SetDO drillDone,1;
WaitUntil drillDone = 0;
        MoveL RelTool(Target_3860,0,0,-10),v30,z10,DrillTool\WObj:=FakeWing;
        MoveL RelTool(Target_3870,0,0,-10),v30,z10,DrillTool\WObj:=FakeWing;
        MoveL Target_3870,v30,fine,DrillTool\WObj:=FakeWing;
SetDO drillDone,1;
WaitUntil drillDone = 0;
        MoveL RelTool(Target_3870,0,0,-10),v30,z10,DrillTool\WObj:=FakeWing;
        MoveL RelTool(Target_3880,0,0,-10),v30,z10,DrillTool\WObj:=FakeWing;
        MoveL Target_3880,v30,fine,DrillTool\WObj:=FakeWing;
SetDO drillDone,1;
WaitUntil drillDone = 0;
        MoveL RelTool(Target_3880,0,0,-10),v30,z10,DrillTool\WObj:=FakeWing;
        MoveL RelTool(Target_3890,0,0,-10),v30,z10,DrillTool\WObj:=FakeWing;
        MoveL Target_3890,v30,fine,DrillTool\WObj:=FakeWing;
SetDO drillDone,1;
WaitUntil drillDone = 0;
        MoveL RelTool(Target_3890,0,0,-10),v30,z10,DrillTool\WObj:=FakeWing;
        MoveL RelTool(Target_3900,0,0,-10),v30,z10,DrillTool\WObj:=FakeWing;
        MoveL Target_3900,v30,fine,DrillTool\WObj:=FakeWing;
SetDO drillDone,1;
WaitUntil drillDone = 0;
        MoveL RelTool(Target_3900,0,0,-10),v30,z10,DrillTool\WObj:=FakeWing;
        MoveL RelTool(Target_3910,0,0,-10),v30,z10,DrillTool\WObj:=FakeWing;
        MoveL Target_3910,v30,fine,DrillTool\WObj:=FakeWing;
SetDO drillDone,1;
WaitUntil drillDone = 0;
        MoveL RelTool(Target_3910,0,0,-10),v30,z10,DrillTool\WObj:=FakeWing;
        MoveL RelTool(Target_3920,0,0,-10),v30,z10,DrillTool\WObj:=FakeWing;
        MoveL Target_3920,v30,fine,DrillTool\WObj:=FakeWing;
SetDO drillDone,1;
WaitUntil drillDone = 0;
        MoveL RelTool(Target_3920,0,0,-10),v30,z10,DrillTool\WObj:=FakeWing;
        MoveL RelTool(Target_3930,0,0,-10),v30,z10,DrillTool\WObj:=FakeWing;
        MoveL Target_3930,v30,fine,DrillTool\WObj:=FakeWing;
SetDO drillDone,1;
WaitUntil drillDone = 0;
        MoveL RelTool(Target_3930,0,0,-10),v30,z10,DrillTool\WObj:=FakeWing;
        MoveL RelTool(Target_3940,0,0,-10),v30,z10,DrillTool\WObj:=FakeWing;
        MoveL Target_3940,v30,fine,DrillTool\WObj:=FakeWing;
SetDO drillDone,1;
WaitUntil drillDone = 0;
        MoveL RelTool(Target_3940,0,0,-10),v30,z10,DrillTool\WObj:=FakeWing;
        MoveL RelTool(Target_3950,0,0,-10),v30,z10,DrillTool\WObj:=FakeWing;
        MoveL Target_3950,v30,fine,DrillTool\WObj:=FakeWing;
SetDO drillDone,1;
WaitUntil drillDone = 0;
        MoveL RelTool(Target_3950,0,0,-10),v30,z10,DrillTool\WObj:=FakeWing;
        MoveL RelTool(Target_3960,0,0,-10),v30,z10,DrillTool\WObj:=FakeWing;
        MoveL Target_3960,v30,fine,DrillTool\WObj:=FakeWing;
SetDO drillDone,1;
WaitUntil drillDone = 0;
        MoveL RelTool(Target_3960,0,0,-10),v30,z10,DrillTool\WObj:=FakeWing;
        MoveL RelTool(Target_3970,0,0,-10),v30,z10,DrillTool\WObj:=FakeWing;
        MoveL Target_3970,v30,fine,DrillTool\WObj:=FakeWing;
SetDO drillDone,1;
WaitUntil drillDone = 0;
        MoveL RelTool(Target_3970,0,0,-10),v30,z10,DrillTool\WObj:=FakeWing;
        MoveL RelTool(Target_3980,0,0,-10),v30,z10,DrillTool\WObj:=FakeWing;
        MoveL Target_3980,v30,fine,DrillTool\WObj:=FakeWing;
SetDO drillDone,1;
WaitUntil drillDone = 0;
        MoveL RelTool(Target_3980,0,0,-10),v30,z10,DrillTool\WObj:=FakeWing;
        MoveL RelTool(Target_3990,0,0,-10),v30,z10,DrillTool\WObj:=FakeWing;
        MoveL Target_3990,v30,fine,DrillTool\WObj:=FakeWing;
SetDO drillDone,1;
WaitUntil drillDone = 0;
        MoveL RelTool(Target_3990,0,0,-10),v30,z10,DrillTool\WObj:=FakeWing;
        MoveL RelTool(Target_4000,0,0,-10),v30,z10,DrillTool\WObj:=FakeWing;
        MoveL Target_4000,v30,fine,DrillTool\WObj:=FakeWing;
SetDO drillDone,1;
WaitUntil drillDone = 0;
        MoveL RelTool(Target_4000,0,0,-10),v30,z10,DrillTool\WObj:=FakeWing;
        MoveL RelTool(Target_4010,0,0,-10),v30,z10,DrillTool\WObj:=FakeWing;
        MoveL Target_4010,v30,fine,DrillTool\WObj:=FakeWing;
SetDO drillDone,1;
WaitUntil drillDone = 0;
        MoveL RelTool(Target_4010,0,0,-10),v30,z10,DrillTool\WObj:=FakeWing;
        MoveL RelTool(Target_4020,0,0,-10),v30,z10,DrillTool\WObj:=FakeWing;
        MoveL Target_4020,v30,fine,DrillTool\WObj:=FakeWing;
SetDO drillDone,1;
WaitUntil drillDone = 0;
        MoveL RelTool(Target_4020,0,0,-10),v30,z10,DrillTool\WObj:=FakeWing;
        MoveL RelTool(Target_4030,0,0,-10),v30,z10,DrillTool\WObj:=FakeWing;
        MoveL Target_4030,v30,fine,DrillTool\WObj:=FakeWing;
SetDO drillDone,1;
WaitUntil drillDone = 0;
        MoveL RelTool(Target_4030,0,0,-10),v30,z10,DrillTool\WObj:=FakeWing;
        MoveL RelTool(Target_4040,0,0,-10),v30,z10,DrillTool\WObj:=FakeWing;
        MoveL Target_4040,v30,fine,DrillTool\WObj:=FakeWing;
SetDO drillDone,1;
WaitUntil drillDone = 0;
        MoveL RelTool(Target_4040,0,0,-10),v30,z10,DrillTool\WObj:=FakeWing;
        MoveL RelTool(Target_4050,0,0,-10),v30,z10,DrillTool\WObj:=FakeWing;
        MoveL Target_4050,v30,fine,DrillTool\WObj:=FakeWing;
SetDO drillDone,1;
WaitUntil drillDone = 0;
        MoveL RelTool(Target_4050,0,0,-10),v30,z10,DrillTool\WObj:=FakeWing;
        MoveL RelTool(Target_4060,0,0,-10),v30,z10,DrillTool\WObj:=FakeWing;
        MoveL Target_4060,v30,fine,DrillTool\WObj:=FakeWing;
SetDO drillDone,1;
WaitUntil drillDone = 0;
        MoveL RelTool(Target_4060,0,0,-10),v30,z10,DrillTool\WObj:=FakeWing;
        MoveL RelTool(Target_4070,0,0,-10),v30,z10,DrillTool\WObj:=FakeWing;
        MoveL Target_4070,v30,fine,DrillTool\WObj:=FakeWing;
SetDO drillDone,1;
WaitUntil drillDone = 0;
        MoveL RelTool(Target_4070,0,0,-10),v30,z10,DrillTool\WObj:=FakeWing;
        MoveL RelTool(Target_4080,0,0,-10),v30,z10,DrillTool\WObj:=FakeWing;
        MoveL Target_4080,v30,fine,DrillTool\WObj:=FakeWing;
SetDO drillDone,1;
WaitUntil drillDone = 0;
        MoveL RelTool(Target_4080,0,0,-10),v30,z10,DrillTool\WObj:=FakeWing;
        MoveL RelTool(Target_4090,0,0,-10),v30,z10,DrillTool\WObj:=FakeWing;
        MoveL Target_4090,v30,fine,DrillTool\WObj:=FakeWing;
SetDO drillDone,1;
WaitUntil drillDone = 0;
        MoveL RelTool(Target_4090,0,0,-10),v30,z10,DrillTool\WObj:=FakeWing;
        MoveL RelTool(Target_4100,0,0,-10),v30,z10,DrillTool\WObj:=FakeWing;
        MoveL Target_4100,v30,fine,DrillTool\WObj:=FakeWing;
SetDO drillDone,1;
WaitUntil drillDone = 0;
        MoveL RelTool(Target_4100,0,0,-10),v30,z10,DrillTool\WObj:=FakeWing;
        MoveL RelTool(Target_4110,0,0,-10),v30,z10,DrillTool\WObj:=FakeWing;
        MoveL Target_4110,v30,fine,DrillTool\WObj:=FakeWing;
SetDO drillDone,1;
WaitUntil drillDone = 0;
        MoveL RelTool(Target_4110,0,0,-10),v30,z10,DrillTool\WObj:=FakeWing;
        MoveL RelTool(Target_4120,0,0,-10),v30,z10,DrillTool\WObj:=FakeWing;
        MoveL Target_4120,v30,fine,DrillTool\WObj:=FakeWing;
SetDO drillDone,1;
WaitUntil drillDone = 0;
        MoveL RelTool(Target_4120,0,0,-10),v30,z10,DrillTool\WObj:=FakeWing;
        MoveL RelTool(Target_4130,0,0,-10),v30,z10,DrillTool\WObj:=FakeWing;
        MoveL Target_4130,v30,fine,DrillTool\WObj:=FakeWing;
SetDO drillDone,1;
WaitUntil drillDone = 0;
        MoveL RelTool(Target_4130,0,0,-10),v30,z10,DrillTool\WObj:=FakeWing;
        MoveL RelTool(Target_4140,0,0,-10),v30,z10,DrillTool\WObj:=FakeWing;
        MoveL Target_4140,v30,fine,DrillTool\WObj:=FakeWing;
SetDO drillDone,1;
WaitUntil drillDone = 0;
        MoveL RelTool(Target_4140,0,0,-10),v30,z10,DrillTool\WObj:=FakeWing;
        MoveL RelTool(Target_4150,0,0,-10),v30,z10,DrillTool\WObj:=FakeWing;
        MoveL Target_4150,v30,fine,DrillTool\WObj:=FakeWing;
SetDO drillDone,1;
WaitUntil drillDone = 0;
        MoveL RelTool(Target_4150,0,0,-10),v30,z10,DrillTool\WObj:=FakeWing;
        MoveL RelTool(Target_4160,0,0,-10),v30,z10,DrillTool\WObj:=FakeWing;
        MoveL Target_4160,v30,fine,DrillTool\WObj:=FakeWing;
SetDO drillDone,1;
WaitUntil drillDone = 0;
        MoveL RelTool(Target_4160,0,0,-10),v30,z10,DrillTool\WObj:=FakeWing;
        MoveL RelTool(Target_4170,0,0,-10),v30,z10,DrillTool\WObj:=FakeWing;
        MoveL Target_4170,v30,fine,DrillTool\WObj:=FakeWing;
SetDO drillDone,1;
WaitUntil drillDone = 0;
        MoveL RelTool(Target_4170,0,0,-10),v30,z10,DrillTool\WObj:=FakeWing;
        MoveL RelTool(Target_4180,0,0,-10),v30,z10,DrillTool\WObj:=FakeWing;
        MoveL Target_4180,v30,fine,DrillTool\WObj:=FakeWing;
SetDO drillDone,1;
WaitUntil drillDone = 0;
        MoveL RelTool(Target_4180,0,0,-10),v30,z10,DrillTool\WObj:=FakeWing;
        MoveL RelTool(Target_4190,0,0,-10),v30,z10,DrillTool\WObj:=FakeWing;
        MoveL Target_4190,v30,fine,DrillTool\WObj:=FakeWing;
SetDO drillDone,1;
WaitUntil drillDone = 0;
        MoveL RelTool(Target_4190,0,0,-10),v30,z10,DrillTool\WObj:=FakeWing;
        MoveL RelTool(Target_4200,0,0,-10),v30,z10,DrillTool\WObj:=FakeWing;
        MoveL Target_4200,v30,fine,DrillTool\WObj:=FakeWing;
SetDO drillDone,1;
WaitUntil drillDone = 0;
        MoveL RelTool(Target_4200,0,0,-10),v30,z10,DrillTool\WObj:=FakeWing;
        MoveL RelTool(Target_4210,0,0,-10),v30,z10,DrillTool\WObj:=FakeWing;
        MoveL Target_4210,v30,fine,DrillTool\WObj:=FakeWing;
SetDO drillDone,1;
WaitUntil drillDone = 0;
        MoveL RelTool(Target_4210,0,0,-10),v30,z10,DrillTool\WObj:=FakeWing;
        MoveL RelTool(Target_4220,0,0,-10),v30,z10,DrillTool\WObj:=FakeWing;
        MoveL Target_4220,v30,fine,DrillTool\WObj:=FakeWing;
SetDO drillDone,1;
WaitUntil drillDone = 0;
        MoveL RelTool(Target_4220,0,0,-10),v30,z10,DrillTool\WObj:=FakeWing;
        MoveL RelTool(Target_4230,0,0,-10),v30,z10,DrillTool\WObj:=FakeWing;
        MoveL Target_4230,v30,fine,DrillTool\WObj:=FakeWing;
SetDO drillDone,1;
WaitUntil drillDone = 0;
        MoveL RelTool(Target_4230,0,0,-10),v30,z10,DrillTool\WObj:=FakeWing;
        MoveL RelTool(Target_4240,0,0,-10),v30,z10,DrillTool\WObj:=FakeWing;
        MoveL Target_4240,v30,fine,DrillTool\WObj:=FakeWing;
SetDO drillDone,1;
WaitUntil drillDone = 0;
        MoveL RelTool(Target_4240,0,0,-10),v30,z10,DrillTool\WObj:=FakeWing;
        MoveL RelTool(Target_4250,0,0,-10),v30,z10,DrillTool\WObj:=FakeWing;
        MoveL Target_4250,v30,fine,DrillTool\WObj:=FakeWing;
SetDO drillDone,1;
WaitUntil drillDone = 0;
        MoveL RelTool(Target_4250,0,0,-10),v30,z10,DrillTool\WObj:=FakeWing;
        MoveL RelTool(Target_4260,0,0,-10),v30,z10,DrillTool\WObj:=FakeWing;
        MoveL Target_4260,v30,fine,DrillTool\WObj:=FakeWing;
SetDO drillDone,1;
WaitUntil drillDone = 0;
        MoveL RelTool(Target_4260,0,0,-10),v30,z10,DrillTool\WObj:=FakeWing;
        MoveL RelTool(Target_4270,0,0,-10),v30,z10,DrillTool\WObj:=FakeWing;
        MoveL Target_4270,v30,fine,DrillTool\WObj:=FakeWing;
SetDO drillDone,1;
WaitUntil drillDone = 0;
        MoveL RelTool(Target_4270,0,0,-10),v30,z10,DrillTool\WObj:=FakeWing;
        MoveL RelTool(Target_4280,0,0,-10),v30,z10,DrillTool\WObj:=FakeWing;
        MoveL Target_4280,v30,fine,DrillTool\WObj:=FakeWing;
SetDO drillDone,1;
WaitUntil drillDone = 0;
        MoveL RelTool(Target_4280,0,0,-10),v30,z10,DrillTool\WObj:=FakeWing;
        MoveL RelTool(Target_4290,0,0,-10),v30,z10,DrillTool\WObj:=FakeWing;
        MoveL Target_4290,v30,fine,DrillTool\WObj:=FakeWing;
SetDO drillDone,1;
WaitUntil drillDone = 0;
        MoveL RelTool(Target_4290,0,0,-10),v30,z10,DrillTool\WObj:=FakeWing;
        MoveL RelTool(Target_4300,0,0,-10),v30,z10,DrillTool\WObj:=FakeWing;
        MoveL Target_4300,v30,fine,DrillTool\WObj:=FakeWing;
SetDO drillDone,1;
WaitUntil drillDone = 0;
        MoveL RelTool(Target_4300,0,0,-10),v30,z10,DrillTool\WObj:=FakeWing;
        MoveL RelTool(Target_4310,0,0,-10),v30,z10,DrillTool\WObj:=FakeWing;
        MoveL Target_4310,v30,fine,DrillTool\WObj:=FakeWing;
SetDO drillDone,1;
WaitUntil drillDone = 0;
        MoveL RelTool(Target_4310,0,0,-10),v30,z10,DrillTool\WObj:=FakeWing;
        MoveL RelTool(Target_4320,0,0,-10),v30,z10,DrillTool\WObj:=FakeWing;
        MoveL Target_4320,v30,fine,DrillTool\WObj:=FakeWing;
SetDO drillDone,1;
WaitUntil drillDone = 0;
        MoveL RelTool(Target_4320,0,0,-10),v30,z10,DrillTool\WObj:=FakeWing;
        MoveL RelTool(Target_4330,0,0,-10),v30,z10,DrillTool\WObj:=FakeWing;
        MoveL Target_4330,v30,fine,DrillTool\WObj:=FakeWing;
SetDO drillDone,1;
WaitUntil drillDone = 0;
        MoveL RelTool(Target_4330,0,0,-10),v30,z10,DrillTool\WObj:=FakeWing;
        MoveL RelTool(Target_4340,0,0,-10),v30,z10,DrillTool\WObj:=FakeWing;
        MoveL Target_4340,v30,fine,DrillTool\WObj:=FakeWing;
SetDO drillDone,1;
WaitUntil drillDone = 0;
        MoveL RelTool(Target_4340,0,0,-10),v30,z10,DrillTool\WObj:=FakeWing;
        MoveL RelTool(Target_4350,0,0,-10),v30,z10,DrillTool\WObj:=FakeWing;
        MoveL Target_4350,v30,fine,DrillTool\WObj:=FakeWing;
SetDO drillDone,1;
WaitUntil drillDone = 0;
        MoveL RelTool(Target_4350,0,0,-10),v30,z10,DrillTool\WObj:=FakeWing;
        MoveL RelTool(Target_4360,0,0,-10),v30,z10,DrillTool\WObj:=FakeWing;
        MoveL Target_4360,v30,fine,DrillTool\WObj:=FakeWing;
SetDO drillDone,1;
WaitUntil drillDone = 0;
        MoveL RelTool(Target_4360,0,0,-10),v30,z10,DrillTool\WObj:=FakeWing;
        MoveL RelTool(Target_4370,0,0,-10),v30,z10,DrillTool\WObj:=FakeWing;
        MoveL Target_4370,v30,fine,DrillTool\WObj:=FakeWing;
SetDO drillDone,1;
WaitUntil drillDone = 0;
        MoveL RelTool(Target_4370,0,0,-10),v30,z10,DrillTool\WObj:=FakeWing;
        MoveL RelTool(Target_4380,0,0,-10),v30,z10,DrillTool\WObj:=FakeWing;
        MoveL Target_4380,v30,fine,DrillTool\WObj:=FakeWing;
SetDO drillDone,1;
WaitUntil drillDone = 0;
        MoveL RelTool(Target_4380,0,0,-10),v30,z10,DrillTool\WObj:=FakeWing;
        MoveL RelTool(Target_4390,0,0,-10),v30,z10,DrillTool\WObj:=FakeWing;
        MoveL Target_4390,v30,fine,DrillTool\WObj:=FakeWing;
SetDO drillDone,1;
WaitUntil drillDone = 0;
        MoveL RelTool(Target_4390,0,0,-10),v30,z10,DrillTool\WObj:=FakeWing;
        MoveL RelTool(Target_4400,0,0,-10),v30,z10,DrillTool\WObj:=FakeWing;
        MoveL Target_4400,v30,fine,DrillTool\WObj:=FakeWing;
SetDO drillDone,1;
WaitUntil drillDone = 0;
        MoveL RelTool(Target_4400,0,0,-10),v30,z10,DrillTool\WObj:=FakeWing;
        MoveL RelTool(Target_4410,0,0,-10),v30,z10,DrillTool\WObj:=FakeWing;
        MoveL Target_4410,v30,fine,DrillTool\WObj:=FakeWing;
SetDO drillDone,1;
WaitUntil drillDone = 0;
        MoveL RelTool(Target_4410,0,0,-10),v30,z10,DrillTool\WObj:=FakeWing;
        MoveL RelTool(Target_4420,0,0,-10),v30,z10,DrillTool\WObj:=FakeWing;
        MoveL Target_4420,v30,fine,DrillTool\WObj:=FakeWing;
SetDO drillDone,1;
WaitUntil drillDone = 0;
        MoveL RelTool(Target_4420,0,0,-10),v30,z10,DrillTool\WObj:=FakeWing;
        MoveL RelTool(Target_4430,0,0,-10),v30,z10,DrillTool\WObj:=FakeWing;
        MoveL Target_4430,v30,fine,DrillTool\WObj:=FakeWing;
SetDO drillDone,1;
WaitUntil drillDone = 0;
        MoveL RelTool(Target_4430,0,0,-10),v30,z10,DrillTool\WObj:=FakeWing;
        MoveL RelTool(Target_4440,0,0,-10),v30,z10,DrillTool\WObj:=FakeWing;
        MoveL Target_4440,v30,fine,DrillTool\WObj:=FakeWing;
SetDO drillDone,1;
WaitUntil drillDone = 0;
        MoveL RelTool(Target_4440,0,0,-10),v30,z10,DrillTool\WObj:=FakeWing;
        MoveL RelTool(Target_4450,0,0,-10),v30,z10,DrillTool\WObj:=FakeWing;
        MoveL Target_4450,v30,fine,DrillTool\WObj:=FakeWing;
SetDO drillDone,1;
WaitUntil drillDone = 0;
        MoveL RelTool(Target_4450,0,0,-10),v30,z10,DrillTool\WObj:=FakeWing;
        MoveL RelTool(Target_4460,0,0,-10),v30,z10,DrillTool\WObj:=FakeWing;
        MoveL Target_4460,v30,fine,DrillTool\WObj:=FakeWing;
SetDO drillDone,1;
WaitUntil drillDone = 0;
        MoveL RelTool(Target_4460,0,0,-10),v30,z10,DrillTool\WObj:=FakeWing;
        MoveL RelTool(Target_4470,0,0,-10),v30,z10,DrillTool\WObj:=FakeWing;
        MoveL Target_4470,v30,fine,DrillTool\WObj:=FakeWing;
SetDO drillDone,1;
WaitUntil drillDone = 0;
        MoveL RelTool(Target_4470,0,0,-10),v30,z10,DrillTool\WObj:=FakeWing;
        MoveL RelTool(Target_4480,0,0,-10),v30,z10,DrillTool\WObj:=FakeWing;
        MoveL Target_4480,v30,fine,DrillTool\WObj:=FakeWing;
SetDO drillDone,1;
WaitUntil drillDone = 0;
        MoveL RelTool(Target_4480,0,0,-10),v30,z10,DrillTool\WObj:=FakeWing;
        MoveL RelTool(Target_4490,0,0,-10),v30,z10,DrillTool\WObj:=FakeWing;
        MoveL Target_4490,v30,fine,DrillTool\WObj:=FakeWing;
SetDO drillDone,1;
WaitUntil drillDone = 0;
        MoveL RelTool(Target_4490,0,0,-10),v30,z10,DrillTool\WObj:=FakeWing;
        MoveL RelTool(Target_4500,0,0,-10),v30,z10,DrillTool\WObj:=FakeWing;
        MoveL Target_4500,v30,fine,DrillTool\WObj:=FakeWing;
SetDO drillDone,1;
WaitUntil drillDone = 0;
        MoveL RelTool(Target_4500,0,0,-10),v30,z10,DrillTool\WObj:=FakeWing;
        MoveL RelTool(Target_4510,0,0,-10),v30,z10,DrillTool\WObj:=FakeWing;
        MoveL Target_4510,v30,fine,DrillTool\WObj:=FakeWing;
SetDO drillDone,1;
WaitUntil drillDone = 0;
        MoveL RelTool(Target_4510,0,0,-10),v30,z10,DrillTool\WObj:=FakeWing;
        MoveL RelTool(Target_4520,0,0,-10),v30,z10,DrillTool\WObj:=FakeWing;
        MoveL Target_4520,v30,fine,DrillTool\WObj:=FakeWing;
SetDO drillDone,1;
WaitUntil drillDone = 0;
        MoveL RelTool(Target_4520,0,0,-10),v30,z10,DrillTool\WObj:=FakeWing;
        MoveL RelTool(Target_4530,0,0,-10),v30,z10,DrillTool\WObj:=FakeWing;
        MoveL Target_4530,v30,fine,DrillTool\WObj:=FakeWing;
SetDO drillDone,1;
WaitUntil drillDone = 0;
        MoveL RelTool(Target_4530,0,0,-10),v30,z10,DrillTool\WObj:=FakeWing;
        MoveL RelTool(Target_4540,0,0,-10),v30,z10,DrillTool\WObj:=FakeWing;
        MoveL Target_4540,v30,fine,DrillTool\WObj:=FakeWing;
SetDO drillDone,1;
WaitUntil drillDone = 0;
        MoveL RelTool(Target_4540,0,0,-10),v30,z10,DrillTool\WObj:=FakeWing;
        MoveL RelTool(Target_4550,0,0,-10),v30,z10,DrillTool\WObj:=FakeWing;
        MoveL Target_4550,v30,fine,DrillTool\WObj:=FakeWing;
SetDO drillDone,1;
WaitUntil drillDone = 0;
        MoveL RelTool(Target_4550,0,0,-10),v30,z10,DrillTool\WObj:=FakeWing;
        MoveL RelTool(Target_4560,0,0,-10),v30,z10,DrillTool\WObj:=FakeWing;
        MoveL Target_4560,v30,fine,DrillTool\WObj:=FakeWing;
SetDO drillDone,1;
WaitUntil drillDone = 0;
        MoveL RelTool(Target_4560,0,0,-10),v30,z10,DrillTool\WObj:=FakeWing;
        MoveL RelTool(Target_4570,0,0,-10),v30,z10,DrillTool\WObj:=FakeWing;
        MoveL Target_4570,v30,fine,DrillTool\WObj:=FakeWing;
SetDO drillDone,1;
WaitUntil drillDone = 0;
        MoveL RelTool(Target_4570,0,0,-10),v30,z10,DrillTool\WObj:=FakeWing;
        MoveL RelTool(Target_4580,0,0,-10),v30,z10,DrillTool\WObj:=FakeWing;
        MoveL Target_4580,v30,fine,DrillTool\WObj:=FakeWing;
SetDO drillDone,1;
WaitUntil drillDone = 0;
        MoveL RelTool(Target_4580,0,0,-10),v30,z10,DrillTool\WObj:=FakeWing;
        MoveL RelTool(Target_4590,0,0,-10),v30,z10,DrillTool\WObj:=FakeWing;
        MoveL Target_4590,v30,fine,DrillTool\WObj:=FakeWing;
SetDO drillDone,1;
WaitUntil drillDone = 0;
        MoveL RelTool(Target_4590,0,0,-10),v30,z10,DrillTool\WObj:=FakeWing;
        MoveL RelTool(Target_4600,0,0,-10),v30,z10,DrillTool\WObj:=FakeWing;
        MoveL Target_4600,v30,fine,DrillTool\WObj:=FakeWing;
SetDO drillDone,1;
WaitUntil drillDone = 0;
        MoveL RelTool(Target_4600,0,0,-10),v30,z10,DrillTool\WObj:=FakeWing;
        MoveL RelTool(Target_4610,0,0,-10),v30,z10,DrillTool\WObj:=FakeWing;
        MoveL Target_4610,v30,fine,DrillTool\WObj:=FakeWing;
SetDO drillDone,1;
WaitUntil drillDone = 0;
        MoveL RelTool(Target_4610,0,0,-10),v30,z10,DrillTool\WObj:=FakeWing;
        MoveL RelTool(Target_4620,0,0,-10),v30,z10,DrillTool\WObj:=FakeWing;
        MoveL Target_4620,v30,fine,DrillTool\WObj:=FakeWing;
SetDO drillDone,1;
WaitUntil drillDone = 0;
        MoveL RelTool(Target_4620,0,0,-10),v30,z10,DrillTool\WObj:=FakeWing;
        MoveL RelTool(Target_4630,0,0,-10),v30,z10,DrillTool\WObj:=FakeWing;
        MoveL Target_4630,v30,fine,DrillTool\WObj:=FakeWing;
SetDO drillDone,1;
WaitUntil drillDone = 0;
        MoveL RelTool(Target_4630,0,0,-10),v30,z10,DrillTool\WObj:=FakeWing;
        MoveL RelTool(Target_4640,0,0,-10),v30,z10,DrillTool\WObj:=FakeWing;
        MoveL Target_4640,v30,fine,DrillTool\WObj:=FakeWing;
SetDO drillDone,1;
WaitUntil drillDone = 0;
        MoveL RelTool(Target_4640,0,0,-10),v30,z10,DrillTool\WObj:=FakeWing;
        MoveL RelTool(Target_4650,0,0,-10),v30,z10,DrillTool\WObj:=FakeWing;
        MoveL Target_4650,v30,fine,DrillTool\WObj:=FakeWing;
SetDO drillDone,1;
WaitUntil drillDone = 0;
        MoveL RelTool(Target_4650,0,0,-10),v30,z10,DrillTool\WObj:=FakeWing;
        MoveL RelTool(Target_4660,0,0,-10),v30,z10,DrillTool\WObj:=FakeWing;
        MoveL Target_4660,v30,fine,DrillTool\WObj:=FakeWing;
SetDO drillDone,1;
WaitUntil drillDone = 0;
        MoveL RelTool(Target_4660,0,0,-10),v30,z10,DrillTool\WObj:=FakeWing;
        MoveL RelTool(Target_4670,0,0,-10),v30,z10,DrillTool\WObj:=FakeWing;
        MoveL Target_4670,v30,fine,DrillTool\WObj:=FakeWing;
SetDO drillDone,1;
WaitUntil drillDone = 0;
        MoveL RelTool(Target_4670,0,0,-10),v30,z10,DrillTool\WObj:=FakeWing;
        MoveL RelTool(Target_4680,0,0,-10),v30,z10,DrillTool\WObj:=FakeWing;
        MoveL Target_4680,v30,fine,DrillTool\WObj:=FakeWing;
SetDO drillDone,1;
WaitUntil drillDone = 0;
        MoveL RelTool(Target_4680,0,0,-10),v30,z10,DrillTool\WObj:=FakeWing;
        MoveL RelTool(Target_4690,0,0,-10),v30,z10,DrillTool\WObj:=FakeWing;
        MoveL Target_4690,v30,fine,DrillTool\WObj:=FakeWing;
SetDO drillDone,1;
WaitUntil drillDone = 0;
        MoveL RelTool(Target_4690,0,0,-10),v30,z10,DrillTool\WObj:=FakeWing;
        MoveL RelTool(Target_4700,0,0,-10),v30,z10,DrillTool\WObj:=FakeWing;
        MoveL Target_4700,v30,fine,DrillTool\WObj:=FakeWing;
SetDO drillDone,1;
WaitUntil drillDone = 0;
        MoveL RelTool(Target_4700,0,0,-10),v30,z10,DrillTool\WObj:=FakeWing;
        MoveL RelTool(Target_4710,0,0,-10),v30,z10,DrillTool\WObj:=FakeWing;
        MoveL Target_4710,v30,fine,DrillTool\WObj:=FakeWing;
SetDO drillDone,1;
WaitUntil drillDone = 0;
        MoveL RelTool(Target_4710,0,0,-10),v30,z10,DrillTool\WObj:=FakeWing;
        MoveL RelTool(Target_4720,0,0,-10),v30,z10,DrillTool\WObj:=FakeWing;
        MoveL Target_4720,v30,fine,DrillTool\WObj:=FakeWing;
SetDO drillDone,1;
WaitUntil drillDone = 0;
        MoveL RelTool(Target_4720,0,0,-10),v30,z10,DrillTool\WObj:=FakeWing;
        MoveL RelTool(Target_4730,0,0,-10),v30,z10,DrillTool\WObj:=FakeWing;
        MoveL Target_4730,v30,fine,DrillTool\WObj:=FakeWing;
SetDO drillDone,1;
WaitUntil drillDone = 0;
        MoveL RelTool(Target_4730,0,0,-10),v30,z10,DrillTool\WObj:=FakeWing;
        MoveL RelTool(Target_4740,0,0,-10),v30,z10,DrillTool\WObj:=FakeWing;
        MoveL Target_4740,v30,fine,DrillTool\WObj:=FakeWing;
SetDO drillDone,1;
WaitUntil drillDone = 0;
        MoveL RelTool(Target_4740,0,0,-10),v30,z10,DrillTool\WObj:=FakeWing;
        MoveL RelTool(Target_4750,0,0,-10),v30,z10,DrillTool\WObj:=FakeWing;
        MoveL Target_4750,v30,fine,DrillTool\WObj:=FakeWing;
SetDO drillDone,1;
WaitUntil drillDone = 0;
        MoveL RelTool(Target_4750,0,0,-10),v30,z10,DrillTool\WObj:=FakeWing;
        MoveL RelTool(Target_4760,0,0,-10),v30,z10,DrillTool\WObj:=FakeWing;
        MoveL Target_4760,v30,fine,DrillTool\WObj:=FakeWing;
SetDO drillDone,1;
WaitUntil drillDone = 0;
        MoveL RelTool(Target_4760,0,0,-10),v30,z10,DrillTool\WObj:=FakeWing;
        MoveL RelTool(Target_4770,0,0,-10),v30,z10,DrillTool\WObj:=FakeWing;
        MoveL Target_4770,v30,fine,DrillTool\WObj:=FakeWing;
SetDO drillDone,1;
WaitUntil drillDone = 0;
        MoveL RelTool(Target_4770,0,0,-10),v30,z10,DrillTool\WObj:=FakeWing;
        MoveL RelTool(Target_4780,0,0,-10),v30,z10,DrillTool\WObj:=FakeWing;
        MoveL Target_4780,v30,fine,DrillTool\WObj:=FakeWing;
SetDO drillDone,1;
WaitUntil drillDone = 0;
        MoveL RelTool(Target_4780,0,0,-10),v30,z10,DrillTool\WObj:=FakeWing;
        MoveL RelTool(Target_4790,0,0,-10),v30,z10,DrillTool\WObj:=FakeWing;
        MoveL Target_4790,v30,fine,DrillTool\WObj:=FakeWing;
SetDO drillDone,1;
WaitUntil drillDone = 0;
        MoveL RelTool(Target_4790,0,0,-10),v30,z10,DrillTool\WObj:=FakeWing;
        MoveL RelTool(Target_4800,0,0,-10),v30,z10,DrillTool\WObj:=FakeWing;
        MoveL Target_4800,v30,fine,DrillTool\WObj:=FakeWing;
SetDO drillDone,1;
WaitUntil drillDone = 0;
        MoveL RelTool(Target_4800,0,0,-10),v30,z10,DrillTool\WObj:=FakeWing;
        MoveL RelTool(Target_4810,0,0,-10),v30,z10,DrillTool\WObj:=FakeWing;
        MoveL Target_4810,v30,fine,DrillTool\WObj:=FakeWing;
SetDO drillDone,1;
WaitUntil drillDone = 0;
        MoveL RelTool(Target_4810,0,0,-10),v30,z10,DrillTool\WObj:=FakeWing;
        MoveL RelTool(Target_4820,0,0,-10),v30,z10,DrillTool\WObj:=FakeWing;
        MoveL Target_4820,v30,fine,DrillTool\WObj:=FakeWing;
SetDO drillDone,1;
WaitUntil drillDone = 0;
        MoveL RelTool(Target_4820,0,0,-10),v30,z10,DrillTool\WObj:=FakeWing;
      ENDPROC
ENDMODULE

--- Backups/Rob2/HOME/Module1.mod ---
MODULE Module1
!PERS tooldata DrillTool:=[TRUE,[[31.792631019,0,229.638935148],[0.945518576,0,0.325568154,0]],[1,[0,0,1],[1,0,0,0],0,0,0]];
PERS tooldata DrillTool:=[TRUE,[[67.056,0,55.372],[0.7071,0,0.7071,0]],[1,[0,0,1],[1,0,0,0],0,0,0]];
PERS wobjdata FakeWing:=[FALSE, TRUE, "",[[154, 596.9, 290],[0, 0.1326, 0, 0.9912]],[[0, 0, 0],[1, 0, 0, 0]]];
!PERS wobjdata FakeWing:=[FALSE, TRUE, "",[[154, 871.22, 290],[0,0,0,1]],[[0, 0, 0],[1, 0, 0, 0]]];
CONST jointtarget jHome:=[[90,0,28.434410486,3.185484116,-20,-3.571881577],[9E+09,9E+09,9E+09,9E+09,9E+09,9E+09]];
	CONST robtarget Target_10:=[[308.4,238.6,-102.8],[-0.0540228184989099,0.529284468395526,0.830894888909729,-0.162951435036297],[0,0,0,1],[9E+09,9E+09,9E+09,9E+09,9E+09,9E+09]];
	CONST robtarget Target_20:=[[308.4,233.9,-101.8],[-0.0547443984118989,0.531632628929442,0.829681024354622,-0.161242663479473],[0,0,0,1],[9E+09,9E+09,9E+09,9E+09,9E+09,9E+09]];
	CONST robtarget Target_30:=[[308.4,229.1,-100.8],[-0.0554746070084852,0.533972825784062,0.828458451488987,-0.159537404573058],[0,0,0,1],[9E+09,9E+09,9E+09,9E+09,9E+09,9E+09]];
	CONST robtarget Target_40:=[[308.4,224.3,-99.8],[-0.05622658655833,0.536260517000348,0.827252679079179,-0.157848768848032],[0,0,0,1],[9E+09,9E+09,9E+09,9E+09,9E+09,9E+09]];
	CONST robtarget Target_50:=[[308.4,219.5,-98.8],[-0.0570173734934169,0.538513452607028,0.826065282156528,-0.156103908012666],[0,0,0,1],[9E+09,9E+09,9E+09,9E+09,9E+09,9E+09]];
	CONST robtarget Target_60:=[[308.4,214.8,-97.9],[-0.0578075887797071,0.540670882363083,0.824917917993721,-0.154414080371918],[0,0,0,1],[9E+09,9E+09,9E+09,9E+09,9E+09,9E+09]];
	CONST robtarget Target_70:=[[308.4,210,-97],[-0.0586053434674626,0.542822347677266,0.823761847214398,-0.15272763879902],[0,0,0,1],[9E+09,9E+09,9E+09,9E+09,9E+09,9E+09]];
	CONST robtarget Target_80:=[[308.4,205.2,-96.1],[-0.0594173744366705,0.544930762338883,0.822621633890505,-0.151042005174497],[0,0,0,1],[9E+09,9E+09,9E+09,9E+09,9E+09,9E+09]];
	CONST robtarget Target_90:=[[308.4,200.4,-95.2],[-0.0602779418746451,0.54700204307425,0.821495947228052,-0.149330985678924],[0,0,0,1],[9E+09,9E+09,9E+09,9E+09,9E+09,9E+09]];
	CONST robtarget Target_100:=[[308.4,195.7,-94.3],[-0.0611233995693708,0.548993739703088,0.820408994029005,-0.147644459117901],[0,0,0,1],[9E+09,9E+09,9E+09,9E+09,9E+09,9E+09]];
	CONST robtarget Target_110:=[[308.4,190.9,-93.5],[-0.0619813474792873,0.550977563261577,0.819312528367716,-0.145976087790734],[0,0,0,1],[9E+09,9E+09,9E+09,9E+09,9E+09,9E+09]];
	CONST robtarget Target_120:=[[308.4,186.1,-92.7],[-0.0628518580764369,0.552923084824419,0.818230272116942,-0.144308447417405],[0,0,0,1],[9E+09,9E+09,9E+09,9E+09,9E+09,9E+09]];
	CONST robtarget Target_130:=[[308.4,181.4,-91.9],[-0.0637401055078415,0.554799250276008,0.817183626452998,-0.142639095272496],[0,0,0,1],[9E+09,9E+09,9E+09,9E+09,9E+09,9E+09]];
	CONST robtarget Target_140:=[[308.4,176.6,-91.1],[-0.0646636661456529,0.55667986221951,0.816127636032455,-0.14093197999016],[0,0,0,1],[9E+09,9E+09,9E+09,9E+09,9E+09,9E+09]];
	CONST robtarget Target_150:=[[308.4,171.8,-90.3],[-0.0655756202077783,0.558514111134058,0.815084460660975,-0.139280823114688],[0,0,0,1],[9E+09,9E+09,9E+09,9E+09,9E+09,9E+09]];
	CONST robtarget Target_160:=[[308.4,167,-89.6],[-0.0664986814080785,0.560314130241802,0.814053991763236,-0.137630299413684],[0,0,0,1],[9E+09,9E+09,9E+09,9E+09,9E+09,9E+09]];
	CONST robtarget Target_170:=[[308.4,162.3,-88.9],[-0.0674308680514497,0.562054271273655,0.813057035081266,-0.135964450801413],[0,0,0,1],[9E+09,9E+09,9E+09,9E+09,9E+09,9E+09]];
	CONST robtarget Target_180:=[[308.4,157.5,-88.2],[-0.0684111361139451,0.563793801471881,0.812048792395899,-0.134287842509463],[0,0,0,1],[9E+09,9E+09,9E+09,9E+09,9E+09,9E+09]];
	CONST robtarget Target_190:=[[308.4,152.7,-87.5],[-0.0693652484196903,0.56549690491479,0.811053916248892,-0.132639578485468],[0,0,0,1],[9E+09,9E+09,9E+09,9E+09,9E+09,9E+09]];
	CONST robtarget Target_200:=[[308.4,148,-86.9],[-0.0703335262208272,0.567141407219054,0.81008981098623,-0.130989760833546],[0,0,0,1],[9E+09,9E+09,9E+09,9E+09,9E+09,9E+09]];
	CONST robtarget Target_210:=[[308.4,143.2,-86.3],[-0.0713134460058373,0.568781437267891,0.809116215699097,-0.129356169280855],[0,0,0,1],[9E+09,9E+09,9E+09,9E+09,9E+09,9E+09]];
	CONST robtarget Target_220:=[[308.4,138.4,-85.7],[-0.0722955709467476,0.570394869197485,0.808154117550502,-0.127710476864027],[0,0,0,1],[9E+09,9E+09,9E+09,9E+09,9E+09,9E+09]];
	CONST robtarget Target_230:=[[308.4,133.6,-85.1],[-0.0733236228418459,0.571984445986194,0.807200120771844,-0.126037315542401],[0,0,0,1],[9E+09,9E+09,9E+09,9E+09,9E+09,9E+09]];
	CONST robtarget Target_240:=[[308.4,128.9,-84.5],[-0.0743414376682748,0.573510671613807,0.806275092793661,-0.124415975385267],[0,0,0,1],[9E+09,9E+09,9E+09,9E+09,9E+09,9E+09]];
	CONST robtarget Target_250:=[[308.4,124.1,-84],[-0.075356372668175,0.575038428608826,0.805342168587324,-0.122785236150173],[0,0,0,1],[9E+09,9E+09,9E+09,9E+09,9E+09,9E+09]];
	CONST robtarget Target_260:=[[308.4,119.3,-83.4],[-0.076379344448792,0.576539662649598,0.804418795175791,-0.121155334597319],[0,0,0,1],[9E+09,9E+09,9E+09,9E+09,9E+09,9E+09]];
	CONST robtarget Target_270:=[[308.4,114.5,-82.9],[-0.0774479655214412,0.578019762866521,0.803501948900264,-0.119497215389307],[0,0,0,1],[9E+09,9E+09,9E+09,9E+09,9E+09,9E+09]];
	CONST robtarget Target_280:=[[308.4,109.8,-82.4],[-0.0784974683762196,0.579443805115183,0.802613049576641,-0.117878398451314],[0,0,0,1],[9E+09,9E+09,9E+09,9E+09,9E+09,9E+09]];
	CONST robtarget Target_290:=[[308.4,105,-82],[-0.0795508130991443,0.58086741275938,0.80171549259436,-0.116262572927284],[0,0,0,1],[9E+09,9E+09,9E+09,9E+09,9E+09,9E+09]];
	CONST robtarget Target_300:=[[308.4,100.2,-81.5],[-0.0806113427211271,0.582266960029181,0.800826422485906,-0.114647458460705],[0,0,0,1],[9E+09,9E+09,9E+09,9E+09,9E+09,9E+09]];
	CONST robtarget Target_310:=[[308.4,95.5,-81.1],[-0.0816819800067539,0.58362055263885,0.799961961293307,-0.11303081510573],[0,0,0,1],[9E+09,9E+09,9E+09,9E+09,9E+09,9E+09]];
	CONST robtarget Target_320:=[[308.4,90.7,-80.7],[-0.082794767336965,0.584978717113686,0.799085584538455,-0.11138741225327],[0,0,0,1],[9E+09,9E+09,9E+09,9E+09,9E+09,9E+09]];
	CONST robtarget Target_330:=[[308.4,85.9,-80.4],[-0.0838836319156044,0.586307668086254,0.798219267880476,-0.109785495509485],[0,0,0,1],[9E+09,9E+09,9E+09,9E+09,9E+09,9E+09]];
	CONST robtarget Target_340:=[[308.4,81.1,-80],[-0.0849789502106103,0.587614708040441,0.797360470344529,-0.108184163571205],[0,0,0,1],[9E+09,9E+09,9E+09,9E+09,9E+09,9E+09]];
	CONST robtarget Target_350:=[[308.4,76.4,-79.7],[-0.0860832915980205,0.588879448289243,0.79652439224517,-0.106581212456363],[0,0,0,1],[9E+09,9E+09,9E+09,9E+09,9E+09,9E+09]];
	CONST robtarget Target_360:=[[308.4,71.6,-79.3],[-0.0872216407657374,0.590150908215717,0.795676956264462,-0.104940326776786],[0,0,0,1],[9E+09,9E+09,9E+09,9E+09,9E+09,9E+09]];
	CONST robtarget Target_370:=[[308.4,66.8,-79],[-0.0883349732594255,0.591395261296902,0.794839102742081,-0.103341076861959],[0,0,0,1],[9E+09,9E+09,9E+09,9E+09,9E+09,9E+09]];
	CONST robtarget Target_380:=[[308.4,62.1,-78.8],[-0.0894651742912847,0.592598007640244,0.794021679272131,-0.101750463270237],[0,0,0,1],[9E+09,9E+09,9E+09,9E+09,9E+09,9E+09]];
	CONST robtarget Target_390:=[[308.4,57.3,-78.5],[-0.090598384829287,0.593801259372321,0.793195720509647,-0.100162597806529],[0,0,0,1],[9E+09,9E+09,9E+09,9E+09,9E+09,9E+09]];
	CONST robtarget Target_400:=[[308.4,52.5,-78.3],[-0.0917370265888429,0.594985280908352,0.792376012395457,-0.0985752932297051],[0,0,0,1],[9E+09,9E+09,9E+09,9E+09,9E+09,9E+09]];
	CONST robtarget Target_410:=[[308.4,47.7,-78.1],[-0.0929120064575001,0.59615659109678,0.791559096194288,-0.0969477961584996],[0,0,0,1],[9E+09,9E+09,9E+09,9E+09,9E+09,9E+09]];
	CONST robtarget Target_420:=[[308.4,43,-77.9],[-0.09406320670459,0.597284763534262,0.790765182273869,-0.0953595873399466],[0,0,0,1],[9E+09,9E+09,9E+09,9E+09,9E+09,9E+09]];
	CONST robtarget Target_430:=[[308.4,38.2,-77.7],[-0.095226295927332,0.59841215591312,0.789961700481073,-0.0937835592863895],[0,0,0,1],[9E+09,9E+09,9E+09,9E+09,9E+09,9E+09]];
	CONST robtarget Target_440:=[[308.4,33.4,-77.5],[-0.0963848720850105,0.599523263975145,0.789164862941784,-0.0921988692111749],[0,0,0,1],[9E+09,9E+09,9E+09,9E+09,9E+09,9E+09]];
	CONST robtarget Target_450:=[[308.4,28.6,-77.4],[-0.0975887713076906,0.600621452045473,0.788368560100788,-0.0905832020964815],[0,0,0,1],[9E+09,9E+09,9E+09,9E+09,9E+09,9E+09]];
	CONST robtarget Target_460:=[[308.4,23.9,-77.3],[-0.0987679840357655,0.601679444358616,0.787594150307987,-0.0890066624835305],[0,0,0,1],[9E+09,9E+09,9E+09,9E+09,9E+09,9E+09]];
	CONST robtarget Target_470:=[[308.4,19.1,-77.2],[-0.0999593935484523,0.602737043222909,0.786810116681356,-0.0874415041968199],[0,0,0,1],[9E+09,9E+09,9E+09,9E+09,9E+09,9E+09]];
	CONST robtarget Target_480:=[[308.4,14.3,-77.1],[-0.101145369475392,0.603779543049934,0.78603214142339,-0.0858682145934034],[0,0,0,1],[9E+09,9E+09,9E+09,9E+09,9E+09,9E+09]];
	CONST robtarget Target_490:=[[308.4,9.6,-77.1],[-0.102337196398047,0.604789512357301,0.785271515729608,-0.0842934787497215],[0,0,0,1],[9E+09,9E+09,9E+09,9E+09,9E+09,9E+09]];
	CONST robtarget Target_500:=[[308.4,4.8,-77.1],[-0.10357270922086,0.605804769828204,0.784497151639023,-0.0826891397240769],[0,0,0,1],[9E+09,9E+09,9E+09,9E+09,9E+09,9E+09]];
	CONST robtarget Target_510:=[[313.1,0,-78.3],[-0.105078931881014,0.603908419748579,0.785960670678543,-0.0807394747199581],[0,0,0,1],[9E+09,9E+09,9E+09,9E+09,9E+09,9E+09]];
	CONST robtarget Target_520:=[[317.8,0,-79.6],[-0.105374424978603,0.601020986689309,0.788170875417063,-0.0803534396509463],[0,0,0,1],[9E+09,9E+09,9E+09,9E+09,9E+09,9E+09]];
	CONST robtarget Target_530:=[[322.6,0,-80.9],[-0.105673526883422,0.598075775645271,0.790408073012287,-0.0799596799601408],[0,0,0,1],[9E+09,9E+09,9E+09,9E+09,9E+09,9E+09]];
	CONST robtarget Target_540:=[[327.3,0,-82.2],[-0.105963764108094,0.595195882921358,0.792578965308918,-0.0795746529954971],[0,0,0,1],[9E+09,9E+09,9E+09,9E+09,9E+09,9E+09]];
	CONST robtarget Target_550:=[[332,0,-83.5],[-0.106251386086706,0.592320277747892,0.7947302963052,-0.079190199254474],[0,0,0,1],[9E+09,9E+09,9E+09,9E+09,9E+09,9E+09]];
	CONST robtarget Target_560:=[[336.7,0,-84.7],[-0.106536384503998,0.589449321136285,0.79686200380534,-0.0788063670024558],[0,0,0,1],[9E+09,9E+09,9E+09,9E+09,9E+09,9E+09]];
	CONST robtarget Target_570:=[[341.4,0,-86],[-0.10681875221387,0.586583368088075,0.798974034358527,-0.0784232037013365],[0,0,0,1],[9E+09,9E+09,9E+09,9E+09,9E+09,9E+09]];
	CONST robtarget Target_580:=[[346.1,0,-87.3],[-0.107098483221086,0.5837227674279,0.801066343122094,-0.0780407559871909],[0,0,0,1],[9E+09,9E+09,9E+09,9E+09,9E+09,9E+09]];
	CONST robtarget Target_590:=[[350.9,0,-88.6],[-0.10738143945292,0.580807183315642,0.80318277565299,-0.0776509572660147],[0,0,0,1],[9E+09,9E+09,9E+09,9E+09,9E+09,9E+09]];
	CONST robtarget Target_600:=[[355.6,0,-89.9],[-0.107655827259247,0.577958440348551,0.80523511878616,-0.0772700948649393],[0,0,0,1],[9E+09,9E+09,9E+09,9E+09,9E+09,9E+09]];
	CONST robtarget Target_610:=[[360.3,0,-91.2],[-0.107927567040378,0.575116064613554,0.807267655440319,-0.0768900837303107],[0,0,0,1],[9E+09,9E+09,9E+09,9E+09,9E+09,9E+09]];
	CONST robtarget Target_620:=[[365,0,-92.4],[-0.108196657225679,0.572280378633997,0.809280373867561,-0.0765109669818548],[0,0,0,1],[9E+09,9E+09,9E+09,9E+09,9E+09,9E+09]];
	CONST robtarget Target_630:=[[369.7,0,-93.7],[-0.108463097290161,0.5694516980844,0.81127327014113,-0.0761327868236447],[0,0,0,1],[9E+09,9E+09,9E+09,9E+09,9E+09,9E+09]];
	CONST robtarget Target_640:=[[374.4,0,-95],[-0.108726887731313,0.566630331689435,0.813246347982093,-0.0757555845305935],[0,0,0,1],[9E+09,9E+09,9E+09,9E+09,9E+09,9E+09]];
	CONST robtarget Target_650:=[[379.1,0,-96.3],[-0.108988030045335,0.563816581133531,0.815199618581601,-0.0753794004363706],[0,0,0,1],[9E+09,9E+09,9E+09,9E+09,9E+09,9E+09]];
	CONST robtarget Target_660:=[[383.9,0,-97.6],[-0.109251997910973,0.560951130314621,0.817174023507502,-0.0749963042807466],[0,0,0,1],[9E+09,9E+09,9E+09,9E+09,9E+09,9E+09]];
	CONST robtarget Target_670:=[[388.6,0,-98.9],[-0.109507796158425,0.558153665430042,0.819087322001568,-0.0746222974976942],[0,0,0,1],[9E+09,9E+09,9E+09,9E+09,9E+09,9E+09]];
	CONST robtarget Target_680:=[[393.3,0,-100.2],[-0.109760956616693,0.555364684329718,0.820980890579095,-0.0742494249533144],[0,0,0,1],[9E+09,9E+09,9E+09,9E+09,9E+09,9E+09]];
	CONST robtarget Target_690:=[[398,0,-101.4],[-0.110011484548332,0.552584459684513,0.822854768602495,-0.0738777231023107],[0,0,0,1],[9E+09,9E+09,9E+09,9E+09,9E+09,9E+09]];
	CONST robtarget Target_700:=[[402.8,4.7,-102.7],[-0.109173771339137,0.548351470788281,0.82567890219086,-0.0751405523856116],[0,0,0,1],[9E+09,9E+09,9E+09,9E+09,9E+09,9E+09]];
	CONST robtarget Target_710:=[[402.8,9.5,-102.8],[-0.108091093958442,0.546903363962133,0.826630501210307,-0.0767791662013001],[0,0,0,1],[9E+09,9E+09,9E+09,9E+09,9E+09,9E+09]];
	CONST robtarget Target_720:=[[402.8,14.2,-102.8],[-0.107022669132324,0.545458796532891,0.827568528802926,-0.0784294569128447],[0,0,0,1],[9E+09,9E+09,9E+09,9E+09,9E+09,9E+09]];
	CONST robtarget Target_730:=[[402.8,19,-102.9],[-0.105962742127289,0.543967513189088,0.828528128312723,-0.0800773530429236],[0,0,0,1],[9E+09,9E+09,9E+09,9E+09,9E+09,9E+09]];
	CONST robtarget Target_740:=[[402.8,23.7,-103],[-0.104896269655517,0.542482047153467,0.829476713310843,-0.0817213754386389],[0,0,0,1],[9E+09,9E+09,9E+09,9E+09,9E+09,9E+09]];
	CONST robtarget Target_750:=[[402.8,28.5,-103.1],[-0.103849243809564,0.540947203735296,0.830446130899949,-0.0833707442958957],[0,0,0,1],[9E+09,9E+09,9E+09,9E+09,9E+09,9E+09]];
	CONST robtarget Target_760:=[[402.8,33.2,-103.2],[-0.102816242063543,0.539415722987032,0.83140180114988,-0.0850326008483989],[0,0,0,1],[9E+09,9E+09,9E+09,9E+09,9E+09,9E+09]];
	CONST robtarget Target_770:=[[402.8,38,-103.4],[-0.101782695272046,0.537835700102673,0.832381528602919,-0.0866835248411941],[0,0,0,1],[9E+09,9E+09,9E+09,9E+09,9E+09,9E+09]];
	CONST robtarget Target_780:=[[402.8,42.7,-103.6],[-0.100763181264532,0.536258987956148,0.833347380044937,-0.0883471748837484],[0,0,0,1],[9E+09,9E+09,9E+09,9E+09,9E+09,9E+09]];
	CONST robtarget Target_790:=[[402.8,47.5,-103.8],[-0.0997439357155413,0.53463218512944,0.834337870776175,-0.0899993961111565],[0,0,0,1],[9E+09,9E+09,9E+09,9E+09,9E+09,9E+09]];
	CONST robtarget Target_800:=[[402.8,52.2,-104],[-0.0987387394706192,0.533008633679001,0.835314349416395,-0.0916645810030375],[0,0,0,1],[9E+09,9E+09,9E+09,9E+09,9E+09,9E+09]];
	CONST robtarget Target_810:=[[402.8,57,-104.2],[-0.0977442049376423,0.531331798074137,0.836314920035596,-0.0933270876126915],[0,0,0,1],[9E+09,9E+09,9E+09,9E+09,9E+09,9E+09]];
	CONST robtarget Target_820:=[[402.8,61.7,-104.5],[-0.0967635456695024,0.529658037088889,0.837301369836592,-0.0950031370344002],[0,0,0,1],[9E+09,9E+09,9E+09,9E+09,9E+09,9E+09]];
	CONST robtarget Target_830:=[[402.8,66.5,-104.8],[-0.0957846493359272,0.527930745779311,0.838313724949949,-0.0966670945722251],[0,0,0,1],[9E+09,9E+09,9E+09,9E+09,9E+09,9E+09]];
	CONST robtarget Target_840:=[[402.8,71.2,-105.1],[-0.0948196695426027,0.526206448577127,0.839311799840147,-0.0983448340929584],[0,0,0,1],[9E+09,9E+09,9E+09,9E+09,9E+09,9E+09]];
	CONST robtarget Target_850:=[[402.8,76,-105.4],[-0.0938665059487625,0.524425036468661,0.84033533676462,-0.10001990787092],[0,0,0,1],[9E+09,9E+09,9E+09,9E+09,9E+09,9E+09]];
	CONST robtarget Target_860:=[[402.8,80.7,-105.7],[-0.0929180477631145,0.522648262706537,0.841345526352199,-0.101699238821492],[0,0,0,1],[9E+09,9E+09,9E+09,9E+09,9E+09,9E+09]];
	CONST robtarget Target_870:=[[402.8,85.5,-106.1],[-0.0919821292202773,0.520812375289864,0.842381870286688,-0.103375733425865],[0,0,0,1],[9E+09,9E+09,9E+09,9E+09,9E+09,9E+09]];
	CONST robtarget Target_880:=[[402.8,90.2,-106.5],[-0.0910511707405547,0.518981138934832,0.843404658938233,-0.10505638018684],[0,0,0,1],[9E+09,9E+09,9E+09,9E+09,9E+09,9E+09]];
	CONST robtarget Target_890:=[[402.8,95,-106.9],[-0.0901423003837138,0.517086668114792,0.844453270290143,-0.106744637503524],[0,0,0,1],[9E+09,9E+09,9E+09,9E+09,9E+09,9E+09]];
	CONST robtarget Target_900:=[[402.8,99.7,-107.3],[-0.0892384702830976,0.515196733091968,0.845488129365696,-0.108437284799062],[0,0,0,1],[9E+09,9E+09,9E+09,9E+09,9E+09,9E+09]];
	CONST robtarget Target_910:=[[402.8,104.5,-107.7],[-0.0883399330737308,0.513245410221675,0.846551620286965,-0.110116117350853],[0,0,0,1],[9E+09,9E+09,9E+09,9E+09,9E+09,9E+09]];
	CONST robtarget Target_920:=[[402.8,109.2,-108.2],[-0.0874639394061394,0.511294325848003,0.847599078876557,-0.111821165915971],[0,0,0,1],[9E+09,9E+09,9E+09,9E+09,9E+09,9E+09]];
	CONST robtarget Target_930:=[[402.8,114,-108.7],[-0.086594071211112,0.509279539964095,0.848675906562912,-0.113512213548427],[0,0,0,1],[9E+09,9E+09,9E+09,9E+09,9E+09,9E+09]];
	CONST robtarget Target_940:=[[402.8,118.7,-109.2],[-0.0857298016167959,0.507269262415874,0.849738515063917,-0.115207432658531],[0,0,0,1],[9E+09,9E+09,9E+09,9E+09,9E+09,9E+09]];
	CONST robtarget Target_950:=[[402.8,123.5,-109.7],[-0.0848894135021422,0.505188317055692,0.850829213294253,-0.116911084122863],[0,0,0,1],[9E+09,9E+09,9E+09,9E+09,9E+09,9E+09]];
	CONST robtarget Target_960:=[[402.8,128.2,-110.3],[-0.0840547505157918,0.503111723230313,0.851905448022469,-0.118619140502658],[0,0,0,1],[9E+09,9E+09,9E+09,9E+09,9E+09,9E+09]];
	CONST robtarget Target_970:=[[402.8,133,-110.9],[-0.0832364492410585,0.500964173166576,0.853011546080285,-0.120324116348267],[0,0,0,1],[9E+09,9E+09,9E+09,9E+09,9E+09,9E+09]];
	CONST robtarget Target_980:=[[402.8,137.7,-111.5],[-0.0824241810789566,0.498820929796159,0.854102914285517,-0.122033381415685],[0,0,0,1],[9E+09,9E+09,9E+09,9E+09,9E+09,9E+09]];
	CONST robtarget Target_990:=[[402.8,142.5,-112.1],[-0.0816371898293487,0.496601394139729,0.855223911280943,-0.123751711699554],[0,0,0,1],[9E+09,9E+09,9E+09,9E+09,9E+09,9E+09]];
	CONST robtarget Target_1000:=[[402.8,147.2,-112.7],[-0.0808485209568348,0.494388693142767,0.85633090303092,-0.125462031172498],[0,0,0,1],[9E+09,9E+09,9E+09,9E+09,9E+09,9E+09]];
	CONST robtarget Target_1010:=[[402.8,152,-113.4],[-0.0800859892650813,0.492096745025681,0.85746829812881,-0.127181545684289],[0,0,0,1],[9E+09,9E+09,9E+09,9E+09,9E+09,9E+09]];
	CONST robtarget Target_1020:=[[402.8,156.7,-114],[-0.0793299911579505,0.48980884043689,0.858590377213851,-0.128905455619714],[0,0,0,1],[9E+09,9E+09,9E+09,9E+09,9E+09,9E+09]];
	CONST robtarget Target_1030:=[[402.8,161.5,-114.7],[-0.0785932462996557,0.487441371392645,0.859744651172031,-0.130625977018442],[0,0,0,1],[9E+09,9E+09,9E+09,9E+09,9E+09,9E+09]];
	CONST robtarget Target_1040:=[[402.8,166.2,-115.5],[-0.0778709701289027,0.485074868994747,0.860882254846597,-0.132363993484447],[0,0,0,1],[9E+09,9E+09,9E+09,9E+09,9E+09,9E+09]];
	CONST robtarget Target_1050:=[[402.8,171,-116.2],[-0.0771614116925029,0.482628601670918,0.862053869763887,-0.134085327384847],[0,0,0,1],[9E+09,9E+09,9E+09,9E+09,9E+09,9E+09]];
	CONST robtarget Target_1060:=[[402.8,175.7,-117],[-0.0764665486570193,0.480183058736185,0.863208454893834,-0.135824373508752],[0,0,0,1],[9E+09,9E+09,9E+09,9E+09,9E+09,9E+09]];
	CONST robtarget Target_1070:=[[402.8,180.5,-117.8],[-0.0757931074196912,0.477651409177404,0.864396792123501,-0.137559884941466],[0,0,0,1],[9E+09,9E+09,9E+09,9E+09,9E+09,9E+09]];
	CONST robtarget Target_1080:=[[402.8,185.2,-118.6],[-0.0751271551758748,0.475123352543578,0.865568767967733,-0.139299742791405],[0,0,0,1],[9E+09,9E+09,9E+09,9E+09,9E+09,9E+09]];
	CONST robtarget Target_1090:=[[402.8,190,-119.4],[-0.0744838693064031,0.47250573765079,0.866775279580614,-0.141035796194364],[0,0,0,1],[9E+09,9E+09,9E+09,9E+09,9E+09,9E+09]];
	CONST robtarget Target_1100:=[[402.8,194.7,-120.2],[-0.0738556750281974,0.469888165079486,0.867963924187749,-0.142790328429366],[0,0,0,1],[9E+09,9E+09,9E+09,9E+09,9E+09,9E+09]];
	CONST robtarget Target_1110:=[[402.8,199.5,-121.1],[-0.0732513409768337,0.467177259971663,0.86918784700694,-0.144541120190431],[0,0,0,1],[9E+09,9E+09,9E+09,9E+09,9E+09,9E+09]];
	CONST robtarget Target_1120:=[[402.8,204.2,-122],[-0.0726551899005905,0.464469513168276,0.870394556627551,-0.146296310653628],[0,0,0,1],[9E+09,9E+09,9E+09,9E+09,9E+09,9E+09]];
	CONST robtarget Target_1130:=[[402.8,209,-122.9],[-0.0720842834673668,0.461664617479993,0.871637303280222,-0.148047453792459],[0,0,0,1],[9E+09,9E+09,9E+09,9E+09,9E+09,9E+09]];
	CONST robtarget Target_1140:=[[402.8,213.7,-123.9],[-0.0715219932106716,0.458862710635186,0.872862376511288,-0.149802833573901],[0,0,0,1],[9E+09,9E+09,9E+09,9E+09,9E+09,9E+09]];
	CONST robtarget Target_1150:=[[402.8,218.5,-124.8],[-0.070993348790441,0.455955857807755,0.874123011714268,-0.15156899600476],[0,0,0,1],[9E+09,9E+09,9E+09,9E+09,9E+09,9E+09]];
	CONST robtarget Target_1160:=[[402.8,223.2,-125.8],[-0.0704667749223318,0.453055520723769,0.875366669396911,-0.153324241014652],[0,0,0,1],[9E+09,9E+09,9E+09,9E+09,9E+09,9E+09]];
	CONST robtarget Target_1170:=[[402.8,228,-126.8],[-0.069975286563823,0.450045871985816,0.87664655423895,-0.155090268294995],[0,0,0,1],[9E+09,9E+09,9E+09,9E+09,9E+09,9E+09]];
	CONST robtarget Target_1180:=[[402.8,232.7,-127.8],[-0.0694932440832772,0.447038675961153,0.877907675075184,-0.156860528067985],[0,0,0,1],[9E+09,9E+09,9E+09,9E+09,9E+09,9E+09]];
	CONST robtarget Target_1190:=[[407.4,232.5,-129.1],[-0.0701438997920973,0.443389919698404,0.879756126929991,-0.156570653575124],[0,0,0,1],[9E+09,9E+09,9E+09,9E+09,9E+09,9E+09]];
	CONST robtarget Target_1200:=[[412.2,232.2,-130.3],[-0.0708036869949546,0.439675185640343,0.881618508706087,-0.156273395518577],[0,0,0,1],[9E+09,9E+09,9E+09,9E+09,9E+09,9E+09]];
	CONST robtarget Target_1210:=[[416.9,231.9,-131.6],[-0.0714627069387675,0.436090821962743,0.883402885516742,-0.155939790873072],[0,0,0,1],[9E+09,9E+09,9E+09,9E+09,9E+09,9E+09]];
	CONST robtarget Target_1220:=[[421.6,231.6,-132.8],[-0.0720886068461626,0.432538296849065,0.885147719252757,-0.155651436304112],[0,0,0,1],[9E+09,9E+09,9E+09,9E+09,9E+09,9E+09]];
	CONST robtarget Target_1230:=[[426.3,231.3,-134.1],[-0.0727050748938696,0.429025989563119,0.886855435467829,-0.155364439126946],[0,0,0,1],[9E+09,9E+09,9E+09,9E+09,9E+09,9E+09]];
	CONST robtarget Target_1240:=[[431,231,-135.3],[-0.0733122343663245,0.425553728621472,0.888526807246585,-0.155078861076456],[0,0,0,1],[9E+09,9E+09,9E+09,9E+09,9E+09,9E+09]];
	CONST robtarget Target_1250:=[[435.7,230.7,-136.6],[-0.0739102097740581,0.42212132118016,0.890162599385395,-0.154794760091252],[0,0,0,1],[9E+09,9E+09,9E+09,9E+09,9E+09,9E+09]];
	CONST robtarget Target_1260:=[[440.5,230.4,-137.8],[-0.0745122120906639,0.418653028889783,0.891799026990306,-0.154505880502683],[0,0,0,1],[9E+09,9E+09,9E+09,9E+09,9E+09,9E+09]];
	CONST robtarget Target_1270:=[[445.2,230.1,-139.1],[-0.0751143593956152,0.415308968869869,0.893367068191316,-0.154180332273884],[0,0,0,1],[9E+09,9E+09,9E+09,9E+09,9E+09,9E+09]];
	CONST robtarget Target_1280:=[[449.9,229.8,-140.3],[-0.0756851876260789,0.411995579065772,0.894899939089706,-0.15390092339393],[0,0,0,1],[9E+09,9E+09,9E+09,9E+09,9E+09,9E+09]];
	CONST robtarget Target_1290:=[[454.6,229.5,-141.6],[-0.0762473421058434,0.40872108006576,0.8964002102088,-0.153623190532203],[0,0,0,1],[9E+09,9E+09,9E+09,9E+09,9E+09,9E+09]];
	CONST robtarget Target_1300:=[[459.3,229.2,-142.8],[-0.0768009502507997,0.405485191721261,0.897868596982472,-0.153347174372641],[0,0,0,1],[9E+09,9E+09,9E+09,9E+09,9E+09,9E+09]];
	CONST robtarget Target_1310:=[[464.1,228.9,-144.1],[-0.0773583028575654,0.402216157514004,0.899337767908794,-0.153066765911142],[0,0,0,1],[9E+09,9E+09,9E+09,9E+09,9E+09,9E+09]];
	CONST robtarget Target_1320:=[[468.8,228.7,-145.3],[-0.0779052718552005,0.39899698285581,0.900770595559414,-0.152789104535194],[0,0,0,1],[9E+09,9E+09,9E+09,9E+09,9E+09,9E+09]];
	CONST robtarget Target_1330:=[[473.5,228.3,-146.6],[-0.0784449698780569,0.395944743888569,0.902122169435086,-0.152478647362774],[0,0,0,1],[9E+09,9E+09,9E+09,9E+09,9E+09,9E+09]];
	CONST robtarget Target_1340:=[[478.2,228.1,-147.8],[-0.0789755718638235,0.392800282298334,0.903495759273722,-0.152204501410216],[0,0,0,1],[9E+09,9E+09,9E+09,9E+09,9E+09,9E+09]];
	CONST robtarget Target_1350:=[[482.9,227.8,-149.1],[-0.079480211101064,0.389757348968478,0.904815847942971,-0.151922303430526],[0,0,0,1],[9E+09,9E+09,9E+09,9E+09,9E+09,9E+09]];
	CONST robtarget Target_1360:=[[487.6,227.5,-150.3],[-0.0799848305294338,0.386747176931651,0.906106578112692,-0.15165723563841],[0,0,0,1],[9E+09,9E+09,9E+09,9E+09,9E+09,9E+09]];
	CONST robtarget Target_1370:=[[492.4,227.2,-151.6],[-0.0804929335251649,0.383706552397799,0.907398364231878,-0.151388169580122],[0,0,0,1],[9E+09,9E+09,9E+09,9E+09,9E+09,9E+09]];
	CONST robtarget Target_1380:=[[497.1,226.9,-152.8],[-0.0810028238309002,0.380777830631852,0.908636966983253,-0.151081595378776],[0,0,0,1],[9E+09,9E+09,9E+09,9E+09,9E+09,9E+09]];
	CONST robtarget Target_1390:=[[497.1,222,-151.8],[-0.0813290537624266,0.384149608847722,0.907488980773307,-0.149259548476051],[0,0,0,1],[9E+09,9E+09,9E+09,9E+09,9E+09,9E+09]];
	CONST robtarget Target_1400:=[[497.1,217.2,-150.8],[-0.0817052988122214,0.387422415146083,0.906369414376248,-0.14738589169808],[0,0,0,1],[9E+09,9E+09,9E+09,9E+09,9E+09,9E+09]];
	CONST robtarget Target_1410:=[[497.1,212.4,-149.8],[-0.0821003495685957,0.390649711482271,0.905250623606648,-0.145511662691714],[0,0,0,1],[9E+09,9E+09,9E+09,9E+09,9E+09,9E+09]];
	CONST robtarget Target_1420:=[[497.1,207.6,-148.8],[-0.0824925655481992,0.393823892416875,0.904131118195996,-0.143682425858401],[0,0,0,1],[9E+09,9E+09,9E+09,9E+09,9E+09,9E+09]];
	CONST robtarget Target_1430:=[[497.1,202.7,-147.9],[-0.0829149781121735,0.397018868118146,0.902989630044964,-0.141812738476147],[0,0,0,1],[9E+09,9E+09,9E+09,9E+09,9E+09,9E+09]];
	CONST robtarget Target_1440:=[[497.1,197.9,-147],[-0.0833723294284235,0.400109234116158,0.901873147936863,-0.139951707710602],[0,0,0,1],[9E+09,9E+09,9E+09,9E+09,9E+09,9E+09]];
	CONST robtarget Target_1450:=[[497.1,193.1,-146.1],[-0.0838469974622208,0.403156804975992,0.90075819436766,-0.138090357728671],[0,0,0,1],[9E+09,9E+09,9E+09,9E+09,9E+09,9E+09]];
	CONST robtarget Target_1460:=[[497.1,188.3,-145.2],[-0.0843167878090531,0.406154114139921,0.899643737945273,-0.136274207525252],[0,0,0,1],[9E+09,9E+09,9E+09,9E+09,9E+09,9E+09]];
	CONST robtarget Target_1470:=[[497.1,183.4,-144.3],[-0.0848168422216677,0.409171395039952,0.898508073561403,-0.134417686714142],[0,0,0,1],[9E+09,9E+09,9E+09,9E+09,9E+09,9E+09]];
	CONST robtarget Target_1480:=[[497.1,178.6,-143.5],[-0.0853496583053356,0.412090385819937,0.897397507883673,-0.132569463248934],[0,0,0,1],[9E+09,9E+09,9E+09,9E+09,9E+09,9E+09]];
	CONST robtarget Target_1490:=[[497.1,173.8,-142.7],[-0.0858677901272042,0.414964306568703,0.896289519475067,-0.130753371550333],[0,0,0,1],[9E+09,9E+09,9E+09,9E+09,9E+09,9E+09]];
	CONST robtarget Target_1500:=[[497.1,169,-141.9],[-0.0864319560074965,0.417803485327623,0.895183340350478,-0.128905204657413],[0,0,0,1],[9E+09,9E+09,9E+09,9E+09,9E+09,9E+09]];
	CONST robtarget Target_1510:=[[497.1,164.1,-141.1],[-0.0870042211294205,0.420653943782027,0.894055790207633,-0.127062067834958],[0,0,0,1],[9E+09,9E+09,9E+09,9E+09,9E+09,9E+09]];
	CONST robtarget Target_1520:=[[497.1,159.3,-140.4],[-0.0875846747965808,0.423404259194089,0.892952775543361,-0.12527209859538],[0,0,0,1],[9E+09,9E+09,9E+09,9E+09,9E+09,9E+09]];
	CONST robtarget Target_1530:=[[497.1,154.5,-139.7],[-0.0881936860705587,0.426127526136662,0.891854024804215,-0.123424485603378],[0,0,0,1],[9E+09,9E+09,9E+09,9E+09,9E+09,9E+09]];
	CONST robtarget Target_1540:=[[497.1,149.6,-139],[-0.0888190416506828,0.428858874632301,0.890733439707747,-0.121594337350781],[0,0,0,1],[9E+09,9E+09,9E+09,9E+09,9E+09,9E+09]];
	CONST robtarget Target_1550:=[[497.1,144.8,-138.3],[-0.089465176247308,0.431504836817279,0.889638798139368,-0.119759621273083],[0,0,0,1],[9E+09,9E+09,9E+09,9E+09,9E+09,9E+09]];
	CONST robtarget Target_1560:=[[497.1,140,-137.6],[-0.0901019068934567,0.434107137934023,0.888546900758733,-0.117970523101938],[0,0,0,1],[9E+09,9E+09,9E+09,9E+09,9E+09,9E+09]];
	CONST robtarget Target_1570:=[[497.1,135.2,-137],[-0.0907750220715357,0.436681615636182,0.887457795723534,-0.116136655465931],[0,0,0,1],[9E+09,9E+09,9E+09,9E+09,9E+09,9E+09]];
	CONST robtarget Target_1580:=[[497.1,130.3,-136.4],[-0.0914643039208925,0.439264011055841,0.886347823416698,-0.114319489256572],[0,0,0,1],[9E+09,9E+09,9E+09,9E+09,9E+09,9E+09]];
	CONST robtarget Target_1590:=[[497.1,125.5,-135.8],[-0.09216351759295,0.441768481872784,0.885264498048338,-0.112486723411854],[0,0,0,1],[9E+09,9E+09,9E+09,9E+09,9E+09,9E+09]];
	CONST robtarget Target_1600:=[[497.1,120.7,-135.3],[-0.0928607089574246,0.444229292117783,0.884183408461757,-0.110710997454669],[0,0,0,1],[9E+09,9E+09,9E+09,9E+09,9E+09,9E+09]];
	CONST robtarget Target_1610:=[[497.1,115.8,-134.7],[-0.0935883247365094,0.446707677832054,0.883082840198059,-0.108895240422325],[0,0,0,1],[9E+09,9E+09,9E+09,9E+09,9E+09,9E+09]];
	CONST robtarget Target_1620:=[[497.1,111,-134.2],[-0.0943426941848549,0.449107069461519,0.882006145432098,-0.107086206551745],[0,0,0,1],[9E+09,9E+09,9E+09,9E+09,9E+09,9E+09]];
	CONST robtarget Target_1630:=[[497.1,106.2,-133.7],[-0.0950757836771643,0.451469158033298,0.880934470350742,-0.105312172376874],[0,0,0,1],[9E+09,9E+09,9E+09,9E+09,9E+09,9E+09]];
	CONST robtarget Target_1640:=[[497.1,101.4,-133.2],[-0.0958534839166685,0.453804683861292,0.879863796394934,-0.103504194698011],[0,0,0,1],[9E+09,9E+09,9E+09,9E+09,9E+09,9E+09]];
	CONST robtarget Target_1650:=[[497.1,96.5,-132.8],[-0.0966377890242803,0.456149949094279,0.878774831163567,-0.101701316546196],[0,0,0,1],[9E+09,9E+09,9E+09,9E+09,9E+09,9E+09]];
	CONST robtarget Target_1660:=[[497.1,91.7,-132.4],[-0.0974138642079185,0.458415825254638,0.877711534519642,-0.0999396437224223],[0,0,0,1],[9E+09,9E+09,9E+09,9E+09,9E+09,9E+09]];
	CONST robtarget Target_1670:=[[497.1,86.9,-132],[-0.0982248398131066,0.460658557283113,0.876650073487825,-0.0981337001204021],[0,0,0,1],[9E+09,9E+09,9E+09,9E+09,9E+09,9E+09]];
	CONST robtarget Target_1680:=[[497.1,82.1,-131.6],[-0.099056043463908,0.462869629811393,0.875590401674392,-0.0963382299360835],[0,0,0,1],[9E+09,9E+09,9E+09,9E+09,9E+09,9E+09]];
	CONST robtarget Target_1690:=[[497.1,77.2,-131.2],[-0.0998935205336521,0.46509010451507,0.874513118442847,-0.094547791666017],[0,0,0,1],[9E+09,9E+09,9E+09,9E+09,9E+09,9E+09]];
	CONST robtarget Target_1700:=[[497.1,72.4,-130.9],[-0.100711100593576,0.467237315650497,0.873462480482747,-0.0927893327375243],[0,0,0,1],[9E+09,9E+09,9E+09,9E+09,9E+09,9E+09]];
	CONST robtarget Target_1710:=[[497.1,67.6,-130.6],[-0.101582810653362,0.4693596378167,0.872410754293778,-0.0910051578807516],[0,0,0,1],[9E+09,9E+09,9E+09,9E+09,9E+09,9E+09]];
	CONST robtarget Target_1720:=[[497.1,62.8,-130.3],[-0.102454384453759,0.471455636967711,0.871363176577917,-0.0892126447406036],[0,0,0,1],[9E+09,9E+09,9E+09,9E+09,9E+09,9E+09]];
	CONST robtarget Target_1730:=[[497.1,57.9,-130],[-0.103306925600619,0.473553916791643,0.870300702751293,-0.0874703024165777],[0,0,0,1],[9E+09,9E+09,9E+09,9E+09,9E+09,9E+09]];
	CONST robtarget Target_1740:=[[497.1,53.1,-129.7],[-0.104207441869202,0.47559319696472,0.869257981542432,-0.0856882814901278],[0,0,0,1],[9E+09,9E+09,9E+09,9E+09,9E+09,9E+09]];
	CONST robtarget Target_1750:=[[497.1,48.3,-129.5],[-0.105117139403384,0.477605783216225,0.868218123595881,-0.0839070479859285],[0,0,0,1],[9E+09,9E+09,9E+09,9E+09,9E+09,9E+09]];
	CONST robtarget Target_1760:=[[497.1,43.4,-129.3],[-0.106032467084069,0.47962714228744,0.86716170499343,-0.0821309789186549],[0,0,0,1],[9E+09,9E+09,9E+09,9E+09,9E+09,9E+09]];
	CONST robtarget Target_1770:=[[497.1,38.6,-129.1],[-0.106934802533463,0.481580560229526,0.866130214185355,-0.0803962940151815],[0,0,0,1],[9E+09,9E+09,9E+09,9E+09,9E+09,9E+09]];
	CONST robtarget Target_1780:=[[497.1,33.8,-128.9],[-0.107881292685985,0.483513693138095,0.865097763106697,-0.0786256669551985],[0,0,0,1],[9E+09,9E+09,9E+09,9E+09,9E+09,9E+09]];
	CONST robtarget Target_1790:=[[497.1,29,-128.8],[-0.108836261807873,0.485421741269383,0.864068044924914,-0.076855806275945],[0,0,0,1],[9E+09,9E+09,9E+09,9E+09,9E+09,9E+09]];
	CONST robtarget Target_1800:=[[497.1,24.1,-128.7],[-0.109796606270312,0.487338272515718,0.863022277739868,-0.0750910215512359],[0,0,0,1],[9E+09,9E+09,9E+09,9E+09,9E+09,9E+09]];
	CONST robtarget Target_1810:=[[497.1,19.3,-128.6],[-0.110742542845466,0.489190564236867,0.862001094207298,-0.0733675313143067],[0,0,0,1],[9E+09,9E+09,9E+09,9E+09,9E+09,9E+09]];
	CONST robtarget Target_1820:=[[497.1,14.5,-128.5],[-0.111721708687057,0.491025084092936,0.860979678217218,-0.0716004210640201],[0,0,0,1],[9E+09,9E+09,9E+09,9E+09,9E+09,9E+09]];
	CONST robtarget Target_1830:=[[497.1,9.7,-128.5],[-0.112719580475348,0.492834933972254,0.859959428792142,-0.0698412833896862],[0,0,0,1],[9E+09,9E+09,9E+09,9E+09,9E+09,9E+09]];
	CONST robtarget Target_1840:=[[497.1,4.8,-128.4],[-0.113685772876722,0.494647900083909,0.858928398856533,-0.0681249266109921],[0,0,0,1],[9E+09,9E+09,9E+09,9E+09,9E+09,9E+09]];
	CONST robtarget Target_1850:=[[501.8,0,-129.7],[-0.114893887892674,0.493878820578874,0.859373763784019,-0.0660290786564159],[0,0,0,1],[9E+09,9E+09,9E+09,9E+09,9E+09,9E+09]];
	CONST robtarget Target_1860:=[[506.5,0,-131],[-0.115086798497098,0.491359540314176,0.860816680506908,-0.0656922637378083],[0,0,0,1],[9E+09,9E+09,9E+09,9E+09,9E+09,9E+09]];
	CONST robtarget Target_1870:=[[511.2,0,-132.3],[-0.115277406305939,0.488853398833187,0.862242372970577,-0.0653572054075515],[0,0,0,1],[9E+09,9E+09,9E+09,9E+09,9E+09,9E+09]];
	CONST robtarget Target_1880:=[[515.9,0,-133.5],[-0.115465730707385,0.48636049319843,0.86365098619319,-0.0650239166424099],[0,0,0,1],[9E+09,9E+09,9E+09,9E+09,9E+09,9E+09]];
	CONST robtarget Target_1890:=[[520.6,0,-134.8],[-0.115651791345235,0.483880914466462,0.865042667104803,-0.0646924096161802],[0,0,0,1],[9E+09,9E+09,9E+09,9E+09,9E+09,9E+09]];
	CONST robtarget Target_1900:=[[525.4,0,-136.1],[-0.115839494861537,0.481362422475873,0.866446636282264,-0.0643557000857994],[0,0,0,1],[9E+09,9E+09,9E+09,9E+09,9E+09,9E+09]];
	CONST robtarget Target_1910:=[[530.1,0,-137.4],[-0.116021040732428,0.478910035122996,0.867804548014806,-0.0640278284082301],[0,0,0,1],[9E+09,9E+09,9E+09,9E+09,9E+09,9E+09]];
	CONST robtarget Target_1920:=[[534.8,0,-138.7],[-0.116200383542556,0.476471214429776,0.86914598147636,-0.063701770523843],[0,0,0,1],[9E+09,9E+09,9E+09,9E+09,9E+09,9E+09]];
	CONST robtarget Target_1930:=[[539.5,0,-140],[-0.116377543768353,0.474046028435897,0.870471089824839,-0.0633775355291968],[0,0,0,1],[9E+09,9E+09,9E+09,9E+09,9E+09,9E+09]];
	CONST robtarget Target_1940:=[[544.2,0,-141.2],[-0.116552542047374,0.471634539747138,0.871780027423315,-0.0630551317943647],[0,0,0,1],[9E+09,9E+09,9E+09,9E+09,9E+09,9E+09]];
	CONST robtarget Target_1950:=[[548.9,0,-142.5],[-0.116725399161056,0.469236805653097,0.873072949711058,-0.0627345669786736],[0,0,0,1],[9E+09,9E+09,9E+09,9E+09,9E+09,9E+09]];
	CONST robtarget Target_1960:=[[553.7,0,-143.8],[-0.116899745834938,0.466802306743809,0.874377013487517,-0.0624090868947495],[0,0,0,1],[9E+09,9E+09,9E+09,9E+09,9E+09,9E+09]];
	CONST robtarget Target_1970:=[[558.4,0,-145.1],[-0.117068339019215,0.464432528270152,0.875638042790104,-0.0620922596028807],[0,0,0,1],[9E+09,9E+09,9E+09,9E+09,9E+09,9E+09]];
	CONST robtarget Target_1980:=[[563.1,0,-146.4],[-0.117234854531426,0.46207664639229,0.87688353169366,-0.0617772902149724],[0,0,0,1],[9E+09,9E+09,9E+09,9E+09,9E+09,9E+09]];
	CONST robtarget Target_1990:=[[567.8,0,-147.7],[-0.117399313568194,0.459734698223149,0.878113638742937,-0.0614641836928336],[0,0,0,1],[9E+09,9E+09,9E+09,9E+09,9E+09,9E+09]];
	CONST robtarget Target_2000:=[[572.5,0,-148.9],[-0.117561737391393,0.457406716158384,0.879328522970735,-0.0611529443675981],[0,0,0,1],[9E+09,9E+09,9E+09,9E+09,9E+09,9E+09]];
	CONST robtarget Target_2010:=[[577.2,0,-150.2],[-0.117722147314052,0.455092727995944,0.880528343792464,-0.0608435759557098],[0,0,0,1],[9E+09,9E+09,9E+09,9E+09,9E+09,9E+09]];
	CONST robtarget Target_2020:=[[582,0,-151.5],[-0.117883913777252,0.452743973942042,0.881738311153518,-0.0605295595215005],[0,0,0,1],[9E+09,9E+09,9E+09,9E+09,9E+09,9E+09]];
	CONST robtarget Target_2030:=[[586.7,0,-152.8],[-0.118040318267545,0.450458338000223,0.882908172474787,-0.0602239816568627],[0,0,0,1],[9E+09,9E+09,9E+09,9E+09,9E+09,9E+09]];
	CONST robtarget Target_2040:=[[586.7,221.3,-176.6],[-0.0891104346648562,0.331098452423926,0.927910467437326,-0.146339706356701],[0,0,0,1],[9E+09,9E+09,9E+09,9E+09,9E+09,9E+09]];
	CONST robtarget Target_2050:=[[582,221.6,-175.3],[-0.0887432500085563,0.333423879444064,0.927077417152281,-0.146562665098053],[0,0,0,1],[9E+09,9E+09,9E+09,9E+09,9E+09,9E+09]];
	CONST robtarget Target_2060:=[[577.2,221.9,-174.1],[-0.0883620433130744,0.335832168276347,0.92620773886212,-0.146792808148981],[0,0,0,1],[9E+09,9E+09,9E+09,9E+09,9E+09,9E+09]];
	CONST robtarget Target_2070:=[[572.5,222.2,-172.8],[-0.0879838114415392,0.338215709016228,0.925340021263495,-0.14701982229259],[0,0,0,1],[9E+09,9E+09,9E+09,9E+09,9E+09,9E+09]];
	CONST robtarget Target_2080:=[[567.8,222.5,-171.6],[-0.0875813502222025,0.340620292727912,0.9244519813159,-0.147295137449658],[0,0,0,1],[9E+09,9E+09,9E+09,9E+09,9E+09,9E+09]];
	CONST robtarget Target_2090:=[[563.1,222.8,-170.3],[-0.0871916700771293,0.34306288786098,0.92354832280148,-0.147526143758382],[0,0,0,1],[9E+09,9E+09,9E+09,9E+09,9E+09,9E+09]];
	CONST robtarget Target_2100:=[[558.4,223.1,-169.1],[-0.0867961732530741,0.345535601674814,0.922626033424251,-0.147759178163931],[0,0,0,1],[9E+09,9E+09,9E+09,9E+09,9E+09,9E+09]];
	CONST robtarget Target_2110:=[[553.7,223.4,-167.8],[-0.0863947561666026,0.348038828247146,0.921684666037846,-0.147994244921791],[0,0,0,1],[9E+09,9E+09,9E+09,9E+09,9E+09,9E+09]];
	CONST robtarget Target_2120:=[[548.9,223.6,-166.6],[-0.0859680323867778,0.350692718960615,0.920678155733562,-0.148242530437806],[0,0,0,1],[9E+09,9E+09,9E+09,9E+09,9E+09,9E+09]];
	CONST robtarget Target_2130:=[[544.2,224,-165.3],[-0.0855449919953143,0.353188933010917,0.919717810856076,-0.148521986039909],[0,0,0,1],[9E+09,9E+09,9E+09,9E+09,9E+09,9E+09]];
	CONST robtarget Target_2140:=[[539.5,224.2,-164.1],[-0.0851149366853577,0.355848342035156,0.918692130954714,-0.148768859462472],[0,0,0,1],[9E+09,9E+09,9E+09,9E+09,9E+09,9E+09]];
	CONST robtarget Target_2150:=[[534.8,224.5,-162.8],[-0.084688474326446,0.358478258694518,0.917669119045982,-0.149012040818775],[0,0,0,1],[9E+09,9E+09,9E+09,9E+09,9E+09,9E+09]];
	CONST robtarget Target_2160:=[[530.1,224.8,-161.6],[-0.0842555477574826,0.36114066646297,0.916624619478424,-0.149257256657101],[0,0,0,1],[9E+09,9E+09,9E+09,9E+09,9E+09,9E+09]];
	CONST robtarget Target_2170:=[[525.4,225.1,-160.3],[-0.0838160442684706,0.363835960211449,0.915558118343285,-0.149504503998719],[0,0,0,1],[9E+09,9E+09,9E+09,9E+09,9E+09,9E+09]];
	CONST robtarget Target_2180:=[[520.6,225.4,-159.1],[-0.0833397223953481,0.366618518161673,0.91444177300152,-0.149805195510177],[0,0,0,1],[9E+09,9E+09,9E+09,9E+09,9E+09,9E+09]];
	CONST robtarget Target_2190:=[[515.9,225.7,-157.8],[-0.0828864355388679,0.369381474041948,0.913329196239681,-0.150056471817903],[0,0,0,1],[9E+09,9E+09,9E+09,9E+09,9E+09,9E+09]];
	CONST robtarget Target_2200:=[[511.2,226,-156.6],[-0.0824262210994575,0.3721784984148,0.912192994594307,-0.15030976018223],[0,0,0,1],[9E+09,9E+09,9E+09,9E+09,9E+09,9E+09]];
	CONST robtarget Target_2210:=[[506.5,226.3,-155.3],[-0.0819589608488699,0.375009977883674,0.911032606747371,-0.15056505128133],[0,0,0,1],[9E+09,9E+09,9E+09,9E+09,9E+09,9E+09]];
	CONST robtarget Target_2220:=[[501.8,226.6,-154.1],[-0.081484535312662,0.377876295599331,0.909847459354232,-0.150822334008115],[0,0,0,1],[9E+09,9E+09,9E+09,9E+09,9E+09,9E+09]];
	CONST robtarget Target_2230:=[[398,233,-126.6],[-0.0688133787721291,0.45083586868829,0.875963745405648,-0.157159966724827],[0,0,0,1],[9E+09,9E+09,9E+09,9E+09,9E+09,9E+09]];
	CONST robtarget Target_2240:=[[393.3,233.3,-125.3],[-0.0681381776210262,0.454591556613989,0.874020583519796,-0.157453882103525],[0,0,0,1],[9E+09,9E+09,9E+09,9E+09,9E+09,9E+09]];
	CONST robtarget Target_2250:=[[388.6,233.6,-124.1],[-0.0674528456392701,0.45838793454485,0.872035529794928,-0.157748692083801],[0,0,0,1],[9E+09,9E+09,9E+09,9E+09,9E+09,9E+09]];
	CONST robtarget Target_2260:=[[383.9,233.9,-122.8],[-0.0667325868025735,0.462216412519589,0.870006349411116,-0.158087639746129],[0,0,0,1],[9E+09,9E+09,9E+09,9E+09,9E+09,9E+09]];
	CONST robtarget Target_2270:=[[379.1,234.2,-121.6],[-0.0660107222946255,0.466180430729295,0.867888740578644,-0.158390418030911],[0,0,0,1],[9E+09,9E+09,9E+09,9E+09,9E+09,9E+09]];
	CONST robtarget Target_2280:=[[374.4,234.5,-120.3],[-0.0652939577196355,0.470099429006276,0.865772248842678,-0.158687236623401],[0,0,0,1],[9E+09,9E+09,9E+09,9E+09,9E+09,9E+09]];
	CONST robtarget Target_2290:=[[369.7,234.8,-119.1],[-0.0645666547616862,0.4740588151663,0.863610618149904,-0.158984549798872],[0,0,0,1],[9E+09,9E+09,9E+09,9E+09,9E+09,9E+09]];
	CONST robtarget Target_2300:=[[365,235.1,-117.8],[-0.0638287234838022,0.478058420378277,0.861403045457561,-0.159282246469257],[0,0,0,1],[9E+09,9E+09,9E+09,9E+09,9E+09,9E+09]];
	CONST robtarget Target_2310:=[[360.3,235.4,-116.6],[-0.0630800791216334,0.482098034826904,0.859148732661681,-0.159580210552165],[0,0,0,1],[9E+09,9E+09,9E+09,9E+09,9E+09,9E+09]];
	CONST robtarget Target_2320:=[[355.6,235.7,-115.3],[-0.0623008583262713,0.4861647259849,0.856844582498321,-0.159936936644151],[0,0,0,1],[9E+09,9E+09,9E+09,9E+09,9E+09,9E+09]];
	CONST robtarget Target_2330:=[[350.9,236,-114.1],[-0.0615302743962089,0.490283545755737,0.854494484540349,-0.160234971164326],[0,0,0,1],[9E+09,9E+09,9E+09,9E+09,9E+09,9E+09]];
	CONST robtarget Target_2340:=[[346.1,236.3,-112.8],[-0.060731418488601,0.4945335001632,0.852041898362416,-0.160539451412005],[0,0,0,1],[9E+09,9E+09,9E+09,9E+09,9E+09,9E+09]];
	CONST robtarget Target_2350:=[[341.4,236.6,-111.6],[-0.0599386765830767,0.49873093242915,0.849591805743821,-0.160837109215425],[0,0,0,1],[9E+09,9E+09,9E+09,9E+09,9E+09,9E+09]];
	CONST robtarget Target_2360:=[[336.7,236.9,-110.3],[-0.0591348869443182,0.502966637218313,0.847091105604348,-0.161134371868289],[0,0,0,1],[9E+09,9E+09,9E+09,9E+09,9E+09,9E+09]];
	CONST robtarget Target_2370:=[[332,237.2,-109.1],[-0.0582930745636434,0.507231486237791,0.844538089294999,-0.161473070686329],[0,0,0,1],[9E+09,9E+09,9E+09,9E+09,9E+09,9E+09]];
	CONST robtarget Target_2380:=[[327.3,237.4,-107.8],[-0.0574580480235626,0.511588011684228,0.841906212830161,-0.161772086023135],[0,0,0,1],[9E+09,9E+09,9E+09,9E+09,9E+09,9E+09]];
	CONST robtarget Target_2390:=[[322.6,237.7,-106.6],[-0.0566207915154303,0.515934486926424,0.839249647066362,-0.162067026464734],[0,0,0,1],[9E+09,9E+09,9E+09,9E+09,9E+09,9E+09]];
	CONST robtarget Target_2400:=[[317.8,238,-105.3],[-0.0557536487314289,0.520413347981774,0.836479714125481,-0.162367378965379],[0,0,0,1],[9E+09,9E+09,9E+09,9E+09,9E+09,9E+09]];
	CONST robtarget Target_2410:=[[313.1,238.3,-104.1],[-0.0548938197151421,0.524831687057051,0.83371461853676,-0.162660086241327],[0,0,0,1],[9E+09,9E+09,9E+09,9E+09,9E+09,9E+09]];
	CONST robtarget Target_2420:=[[209.3,244.8,-76.6],[-0.0330646930109029,0.629121636933686,0.758080962202085,-0.168599960749507],[0,0,0,1],[9E+09,9E+09,9E+09,9E+09,9E+09,9E+09]];
	CONST robtarget Target_2430:=[[204.6,245.1,-75.3],[-0.0319737541914932,0.634010595270966,0.753996912722801,-0.168810247708907],[0,0,0,1],[9E+09,9E+09,9E+09,9E+09,9E+09,9E+09]];
	CONST robtarget Target_2440:=[[199.9,245.4,-74.1],[-0.0308755214603676,0.638899471183747,0.749858816733182,-0.169014564056447],[0,0,0,1],[9E+09,9E+09,9E+09,9E+09,9E+09,9E+09]];
	CONST robtarget Target_2450:=[[195.2,245.7,-72.8],[-0.0297703457473825,0.643786183416851,0.745667572952535,-0.169212727661727],[0,0,0,1],[9E+09,9E+09,9E+09,9E+09,9E+09,9E+09]];
	CONST robtarget Target_2460:=[[190.5,245.9,-71.6],[-0.0286561087187912,0.648679495354103,0.741414655653978,-0.169404982576479],[0,0,0,1],[9E+09,9E+09,9E+09,9E+09,9E+09,9E+09]];
	CONST robtarget Target_2470:=[[185.8,246.3,-70.3],[-0.0275064663910176,0.653536001923108,0.737130270216193,-0.169626216216841],[0,0,0,1],[9E+09,9E+09,9E+09,9E+09,9E+09,9E+09]];
	CONST robtarget Target_2480:=[[181.1,246.5,-69.1],[-0.0263806014436528,0.658411567480971,0.732778649310888,-0.169804955136279],[0,0,0,1],[9E+09,9E+09,9E+09,9E+09,9E+09,9E+09]];
	CONST robtarget Target_2490:=[[176.3,246.8,-67.8],[-0.0252273343467782,0.663370599750435,0.728292378420498,-0.169980118023016],[0,0,0,1],[9E+09,9E+09,9E+09,9E+09,9E+09,9E+09]];
	CONST robtarget Target_2500:=[[171.6,247.1,-66.6],[-0.0240931772944183,0.668212823778592,0.723852169449314,-0.170144578900482],[0,0,0,1],[9E+09,9E+09,9E+09,9E+09,9E+09,9E+09]];
	CONST robtarget Target_2510:=[[166.9,247.4,-65.3],[-0.0229544688497021,0.673040027567628,0.719366014189164,-0.170301941507402],[0,0,0,1],[9E+09,9E+09,9E+09,9E+09,9E+09,9E+09]];
	CONST robtarget Target_2520:=[[162.2,247.7,-64.1],[-0.0218116442228955,0.67785006818605,0.714835383944307,-0.170452078595881],[0,0,0,1],[9E+09,9E+09,9E+09,9E+09,9E+09,9E+09]];
	CONST robtarget Target_2530:=[[157.5,248,-62.8],[-0.020665147486378,0.682640814131333,0.710261824935529,-0.170594872726963],[0,0,0,1],[9E+09,9E+09,9E+09,9E+09,9E+09,9E+09]];
	CONST robtarget Target_2540:=[[152.7,248.3,-61.6],[-0.0194551004124707,0.687502714644314,0.705549371656042,-0.170767680140021],[0,0,0,1],[9E+09,9E+09,9E+09,9E+09,9E+09,9E+09]];
	CONST robtarget Target_2550:=[[148,248.6,-60.3],[-0.0183023566454308,0.692247946763705,0.700894199354632,-0.170895070887628],[0,0,0,1],[9E+09,9E+09,9E+09,9E+09,9E+09,9E+09]];
	CONST robtarget Target_2560:=[[143.3,248.9,-59.1],[-0.0171473278292349,0.696967568679161,0.696201196994802,-0.171014825850804],[0,0,0,1],[9E+09,9E+09,9E+09,9E+09,9E+09,9E+09]];
	CONST robtarget Target_2570:=[[138.6,249.2,-57.8],[-0.0159904837570115,0.701659547870884,0.691472181196874,-0.17112687089315],[0,0,0,1],[9E+09,9E+09,9E+09,9E+09,9E+09,9E+09]];
	CONST robtarget Target_2580:=[[133.9,249.5,-56.6],[-0.0148322979384848,0.706321889232599,0.68670902664697,-0.171231143342349],[0,0,0,1],[9E+09,9E+09,9E+09,9E+09,9E+09,9E+09]];
	CONST robtarget Target_2590:=[[129.2,249.8,-55.3],[-0.0136732464916139,0.710952639941439,0.681913661872113,-0.171327592181889],[0,0,0,1],[9E+09,9E+09,9E+09,9E+09,9E+09,9E+09]];
	CONST robtarget Target_2600:=[[124.4,250.1,-54.1],[-0.0124892710517159,0.715646802561406,0.676985636827823,-0.171417967614427],[0,0,0,1],[9E+09,9E+09,9E+09,9E+09,9E+09,9E+09]];
	CONST robtarget Target_2610:=[[25.4,4.7,0],[-0.0816486492100062,0.771496504751779,0.622277235046125,-0.104391972782008],[0,0,0,1],[9E+09,9E+09,9E+09,9E+09,9E+09,9E+09]];
	CONST robtarget Target_2620:=[[25.4,9.5,0],[-0.0799992230274888,0.771850747246867,0.621828447919395,-0.105716269550184],[0,0,0,1],[9E+09,9E+09,9E+09,9E+09,9E+09,9E+09]];
	CONST robtarget Target_2630:=[[25.4,14.2,-0.1],[-0.0783956408178687,0.772201769929318,0.621374495212959,-0.107015357391473],[0,0,0,1],[9E+09,9E+09,9E+09,9E+09,9E+09,9E+09]];
	CONST robtarget Target_2640:=[[25.4,19,-0.2],[-0.0767785359193531,0.772570517222499,0.620894717021794,-0.108303290416625],[0,0,0,1],[9E+09,9E+09,9E+09,9E+09,9E+09,9E+09]];
	CONST robtarget Target_2650:=[[25.4,23.7,-0.2],[-0.0751268762924455,0.772926904927033,0.620420125378589,-0.109630379565486],[0,0,0,1],[9E+09,9E+09,9E+09,9E+09,9E+09,9E+09]];
	CONST robtarget Target_2660:=[[25.4,28.5,-0.3],[-0.0735091429764661,0.773304826213177,0.619912706592075,-0.110924694545269],[0,0,0,1],[9E+09,9E+09,9E+09,9E+09,9E+09,9E+09]];
	CONST robtarget Target_2670:=[[25.4,33.2,-0.5],[-0.0718893502838438,0.773676551204279,0.619406337541587,-0.112215437644457],[0,0,0,1],[9E+09,9E+09,9E+09,9E+09,9E+09,9E+09]];
	CONST robtarget Target_2680:=[[25.4,37.9,-0.6],[-0.0702251950846496,0.774048910249563,0.618891208798363,-0.113535801353087],[0,0,0,1],[9E+09,9E+09,9E+09,9E+09,9E+09,9E+09]];
	CONST robtarget Target_2690:=[[25.4,42.7,-0.8],[-0.0685947840793333,0.774444127586446,0.618341874516178,-0.114823233989456],[0,0,0,1],[9E+09,9E+09,9E+09,9E+09,9E+09,9E+09]];
	CONST robtarget Target_2700:=[[25.4,47.4,-0.9],[-0.0669689070708674,0.774831453886875,0.617792784809483,-0.116118295675694],[0,0,0,1],[9E+09,9E+09,9E+09,9E+09,9E+09,9E+09]];
	CONST robtarget Target_2710:=[[25.4,52.2,-1.1],[-0.0652893578640036,0.775234130977816,0.61721871302553,-0.117432543223271],[0,0,0,1],[9E+09,9E+09,9E+09,9E+09,9E+09,9E+09]];
	CONST robtarget Target_2720:=[[25.4,56.9,-1.4],[-0.063654337047,0.775633930210214,0.616640125167891,-0.118722734615959],[0,0,0,1],[9E+09,9E+09,9E+09,9E+09,9E+09,9E+09]];
	CONST robtarget Target_2730:=[[25.4,61.7,-1.6],[-0.0619717124676495,0.776047982126195,0.616034600462907,-0.120043356018546],[0,0,0,1],[9E+09,9E+09,9E+09,9E+09,9E+09,9E+09]];
	CONST robtarget Target_2740:=[[25.4,66.4,-1.9],[-0.0603271872625083,0.776461071687208,0.615425263134368,-0.121328397860276],[0,0,0,1],[9E+09,9E+09,9E+09,9E+09,9E+09,9E+09]];
	CONST robtarget Target_2750:=[[25.4,71.2,-2.1],[-0.0586751876109112,0.776894569887548,0.614783164526675,-0.122612031435063],[0,0,0,1],[9E+09,9E+09,9E+09,9E+09,9E+09,9E+09]];
	CONST robtarget Target_2760:=[[25.4,75.9,-2.4],[-0.0569860150022066,0.77731443415222,0.614145686708351,-0.123935225219912],[0,0,0,1],[9E+09,9E+09,9E+09,9E+09,9E+09,9E+09]];
	CONST robtarget Target_2770:=[[25.4,80.7,-2.7],[-0.0553238489574246,0.77776300170738,0.613470169447094,-0.125213162687542],[0,0,0,1],[9E+09,9E+09,9E+09,9E+09,9E+09,9E+09]];
	CONST robtarget Target_2780:=[[25.4,85.4,-3.1],[-0.0536646621305004,0.778203412489929,0.612794807637811,-0.126499314462914],[0,0,0,1],[9E+09,9E+09,9E+09,9E+09,9E+09,9E+09]];
	CONST robtarget Target_2790:=[[25.4,90.1,-3.4],[-0.0520001006783575,0.778651616514941,0.612102328073387,-0.127782587214575],[0,0,0,1],[9E+09,9E+09,9E+09,9E+09,9E+09,9E+09]];
	CONST robtarget Target_2800:=[[25.4,94.9,-3.8],[-0.0502864189787529,0.779116692721743,0.611377853226394,-0.129095219791102],[0,0,0,1],[9E+09,9E+09,9E+09,9E+09,9E+09,9E+09]];
	CONST robtarget Target_2810:=[[25.4,99.6,-4.2],[-0.04861077072326,0.779581431143657,0.610649531901286,-0.130372291436634],[0,0,0,1],[9E+09,9E+09,9E+09,9E+09,9E+09,9E+09]];
	CONST robtarget Target_2820:=[[25.4,104.4,-4.6],[-0.046885611949136,0.780063932790252,0.609887552842283,-0.131678293731398],[0,0,0,1],[9E+09,9E+09,9E+09,9E+09,9E+09,9E+09]];
	CONST robtarget Target_2830:=[[25.4,109.1,-5],[-0.0452028740439187,0.780544008668363,0.609121417468522,-0.132961834716695],[0,0,0,1],[9E+09,9E+09,9E+09,9E+09,9E+09,9E+09]];
	CONST robtarget Target_2840:=[[25.4,113.9,-5.4],[-0.0435063932859472,0.781051177343454,0.608316177335671,-0.134229953830614],[0,0,0,1],[9E+09,9E+09,9E+09,9E+09,9E+09,9E+09]];
	CONST robtarget Target_2850:=[[25.4,118.6,-5.9],[-0.0417706616179563,0.781543829458959,0.607514638958406,-0.135537514784141],[0,0,0,1],[9E+09,9E+09,9E+09,9E+09,9E+09,9E+09]];
	CONST robtarget Target_2860:=[[25.4,123.4,-6.4],[-0.0400656367387652,0.782068484600279,0.606668087171559,-0.136811776376679],[0,0,0,1],[9E+09,9E+09,9E+09,9E+09,9E+09,9E+09]];
	CONST robtarget Target_2870:=[[25.4,128.1,-6.9],[-0.0383577272294432,0.782587224758595,0.605821324762428,-0.138081290801936],[0,0,0,1],[9E+09,9E+09,9E+09,9E+09,9E+09,9E+09]];
	CONST robtarget Target_2880:=[[25.4,132.9,-7.4],[-0.0365986103919072,0.783126667075213,0.604935351521993,-0.139378569055698],[0,0,0,1],[9E+09,9E+09,9E+09,9E+09,9E+09,9E+09]];
	CONST robtarget Target_2890:=[[25.4,137.6,-8],[-0.034877347640361,0.783666646083767,0.604045100801052,-0.140640231212982],[0,0,0,1],[9E+09,9E+09,9E+09,9E+09,9E+09,9E+09]];
	CONST robtarget Target_2900:=[[25.4,142.3,-8.5],[-0.0331524140005,0.784214983247709,0.603132486603527,-0.1419118779355],[0,0,0,1],[9E+09,9E+09,9E+09,9E+09,9E+09,9E+09]];
	CONST robtarget Target_2910:=[[25.4,147.1,-9.1],[-0.0313751328555289,0.784785659070614,0.602177510654819,-0.143210739879962],[0,0,0,1],[9E+09,9E+09,9E+09,9E+09,9E+09,9E+09]];
	CONST robtarget Target_2920:=[[25.4,151.8,-9.7],[-0.0296325952340913,0.785359970763115,0.601217933569803,-0.144459759022046],[0,0,0,1],[9E+09,9E+09,9E+09,9E+09,9E+09,9E+09]];
	CONST robtarget Target_2930:=[[25.4,156.6,-10.3],[-0.0278809945750648,0.78596193798026,0.600210217810398,-0.145719513531353],[0,0,0,1],[9E+09,9E+09,9E+09,9E+09,9E+09,9E+09]];
	CONST robtarget Target_2940:=[[25.4,161.3,-11],[-0.0260874898804154,0.78654858525833,0.5992047460239,-0.147018496259117],[0,0,0,1],[9E+09,9E+09,9E+09,9E+09,9E+09,9E+09]];
	CONST robtarget Target_2950:=[[25.4,166.1,-11.6],[-0.0243197129064465,0.787176744880257,0.598145161875128,-0.148268975882507],[0,0,0,1],[9E+09,9E+09,9E+09,9E+09,9E+09,9E+09]];
	CONST robtarget Target_2960:=[[25.4,170.8,-12.3],[-0.0225484722456159,0.787799513101417,0.597083852612889,-0.149513766943077],[0,0,0,1],[9E+09,9E+09,9E+09,9E+09,9E+09,9E+09]];
	CONST robtarget Target_2970:=[[25.4,175.6,-13],[-0.0207248929133501,0.788445598386254,0.595972909516474,-0.150798900266347],[0,0,0,1],[9E+09,9E+09,9E+09,9E+09,9E+09,9E+09]];
	CONST robtarget Target_2980:=[[25.4,180.3,-13.7],[-0.0189383920181083,0.7890933742209,0.594856495857871,-0.152048457421108],[0,0,0,1],[9E+09,9E+09,9E+09,9E+09,9E+09,9E+09]];
	CONST robtarget Target_2990:=[[25.4,185.1,-14.4],[-0.0170965714657476,0.789768956804693,0.593687446554438,-0.153322920385096],[0,0,0,1],[9E+09,9E+09,9E+09,9E+09,9E+09,9E+09]];
	CONST robtarget Target_3000:=[[25.4,189.8,-15.2],[-0.0152917657314588,0.790446591060719,0.592512479634857,-0.154561670728084],[0,0,0,1],[9E+09,9E+09,9E+09,9E+09,9E+09,9E+09]];
	CONST robtarget Target_3010:=[[25.4,194.5,-16],[-0.0134775760488848,0.791139740266602,0.591307245188397,-0.155794762756806],[0,0,0,1],[9E+09,9E+09,9E+09,9E+09,9E+09,9E+09]];
	CONST robtarget Target_3020:=[[25.4,199.3,-16.8],[-0.0116479972262109,0.79187063814985,0.590041679393542,-0.157022397049646],[0,0,0,1],[9E+09,9E+09,9E+09,9E+09,9E+09,9E+09]];
	CONST robtarget Target_3030:=[[25.4,204,-17.6],[-0.00977383985694139,0.792585828477493,0.588775847716777,-0.158288274033445],[0,0,0,1],[9E+09,9E+09,9E+09,9E+09,9E+09,9E+09]];
	CONST robtarget Target_3040:=[[25.4,208.8,-18.4],[-0.00792422315599783,0.793348049062693,0.587443386601589,-0.159519112566011],[0,0,0,1],[9E+09,9E+09,9E+09,9E+09,9E+09,9E+09]];
	CONST robtarget Target_3050:=[[25.4,213.5,-19.2],[-0.00606983909444402,0.794105676665045,0.586106608579309,-0.160743194945786],[0,0,0,1],[9E+09,9E+09,9E+09,9E+09,9E+09,9E+09]];
	CONST robtarget Target_3060:=[[25.4,218.3,-20.1],[-0.00415671334714131,0.794897215588351,0.584705500460769,-0.161989555573681],[0,0,0,1],[9E+09,9E+09,9E+09,9E+09,9E+09,9E+09]];
	CONST robtarget Target_3070:=[[25.4,223,-21],[-0.00227982923064156,0.795692138630642,0.58329634877276,-0.163199854192462],[0,0,0,1],[9E+09,9E+09,9E+09,9E+09,9E+09,9E+09]];
	CONST robtarget Target_3080:=[[25.4,227.8,-21.9],[-0.000343161028673128,0.796523037582201,0.581818895966585,-0.164431460303543],[0,0,0,1],[9E+09,9E+09,9E+09,9E+09,9E+09,9E+09]];
	CONST robtarget Target_3090:=[[25.4,232.5,-22.9],[0.00155774511334554,0.797353967904281,0.580333117220716,-0.165643280438256],[0,0,0,1],[9E+09,9E+09,9E+09,9E+09,9E+09,9E+09]];
	CONST robtarget Target_3100:=[[25.4,237.3,-23.8],[0.00347861493687028,0.798230983744147,0.578772117197483,-0.166847331964629],[0,0,0,1],[9E+09,9E+09,9E+09,9E+09,9E+09,9E+09]];
	CONST robtarget Target_3110:=[[25.4,242,-24.8],[0.00544599211880825,0.799100144747581,0.577206071085835,-0.168054905718017],[0,0,0,1],[9E+09,9E+09,9E+09,9E+09,9E+09,9E+09]];
	CONST robtarget Target_3120:=[[25.4,246.7,-25.8],[0.00738585622544953,0.799995428854368,0.575595110655205,-0.169242522817864],[0,0,0,1],[9E+09,9E+09,9E+09,9E+09,9E+09,9E+09]];
	CONST robtarget Target_3130:=[[25.4,251.5,-26.8],[0.00934854871281768,0.800936484340026,0.573902636486851,-0.170438013727704],[0,0,0,1],[9E+09,9E+09,9E+09,9E+09,9E+09,9E+09]];
	CONST robtarget Target_3140:=[[25.4,256.2,-27.8],[0.0113580960105811,0.801870156996903,0.57220314404859,-0.171635680770881],[0,0,0,1],[9E+09,9E+09,9E+09,9E+09,9E+09,9E+09]];
	CONST robtarget Target_3150:=[[30.1,255.9,-29.1],[0.0102514536764731,0.798311972467211,0.577166044876818,-0.171674864072409],[0,0,0,1],[9E+09,9E+09,9E+09,9E+09,9E+09,9E+09]];
	CONST robtarget Target_3160:=[[34.8,255.7,-30.3],[0.00918587623296491,0.794714822430291,0.582109096091815,-0.17173517675361],[0,0,0,1],[9E+09,9E+09,9E+09,9E+09,9E+09,9E+09]];
	CONST robtarget Target_3170:=[[39.5,255.3,-31.6],[0.00809672271399045,0.791007704806005,0.58713666184354,-0.171789971587557],[0,0,0,1],[9E+09,9E+09,9E+09,9E+09,9E+09,9E+09]];
	CONST robtarget Target_3180:=[[44.2,255.1,-32.8],[0.0070151140987902,0.787295902256136,0.592104560896076,-0.171837537898278],[0,0,0,1],[9E+09,9E+09,9E+09,9E+09,9E+09,9E+09]];
	CONST robtarget Target_3190:=[[49,254.8,-34.1],[0.00589567441362501,0.783422434180185,0.597220175786478,-0.171879586571441],[0,0,0,1],[9E+09,9E+09,9E+09,9E+09,9E+09,9E+09]];
	CONST robtarget Target_3200:=[[53.7,254.5,-35.3],[0.00479206590257211,0.779572065269462,0.60223753104132,-0.171913895195084],[0,0,0,1],[9E+09,9E+09,9E+09,9E+09,9E+09,9E+09]];
	CONST robtarget Target_3210:=[[58.4,254.2,-36.6],[0.00368184764794892,0.775666917664595,0.607258990533648,-0.171941255243348],[0,0,0,1],[9E+09,9E+09,9E+09,9E+09,9E+09,9E+09]];
	CONST robtarget Target_3220:=[[63.1,253.9,-37.8],[0.00252541762663588,0.771716168657379,0.612280378113319,-0.171931718644344],[0,0,0,1],[9E+09,9E+09,9E+09,9E+09,9E+09,9E+09]];
	CONST robtarget Target_3230:=[[67.8,253.6,-39.1],[0.0014032710037228,0.767703754987846,0.617303856271264,-0.171944538850982],[0,0,0,1],[9E+09,9E+09,9E+09,9E+09,9E+09,9E+09]];
	CONST robtarget Target_3240:=[[72.6,253.3,-40.3],[0.00025194861916876,0.763553257561029,0.622430340887841,-0.171950080349153],[0,0,0,1],[9E+09,9E+09,9E+09,9E+09,9E+09,9E+09]];
	CONST robtarget Target_3250:=[[77.3,253,-41.6],[-0.0008808921358361,0.759436013773593,0.627447246685718,-0.171948008535231],[0,0,0,1],[9E+09,9E+09,9E+09,9E+09,9E+09,9E+09]];
	CONST robtarget Target_3260:=[[82,252.7,-42.8],[-0.00201839954074666,0.755268500999825,0.63245758576152,-0.171938418259215],[0,0,0,1],[9E+09,9E+09,9E+09,9E+09,9E+09,9E+09]];
	CONST robtarget Target_3270:=[[86.7,252.4,-44.1],[-0.00316015182200857,0.751051866701647,0.637459175095774,-0.171921223386319],[0,0,0,1],[9E+09,9E+09,9E+09,9E+09,9E+09,9E+09]];
	CONST robtarget Target_3280:=[[91.4,252.1,-45.3],[-0.00430540759594907,0.74679156851643,0.642449494845078,-0.171879211167342],[0,0,0,1],[9E+09,9E+09,9E+09,9E+09,9E+09,9E+09]];
	CONST robtarget Target_3290:=[[96.1,251.8,-46.6],[-0.00549276498109347,0.742488988783896,0.647425326252885,-0.171814952765686],[0,0,0,1],[9E+09,9E+09,9E+09,9E+09,9E+09,9E+09]];
	CONST robtarget Target_3300:=[[100.9,251.5,-47.8],[-0.00666858886590735,0.738040426737729,0.652491976992652,-0.171773334320405],[0,0,0,1],[9E+09,9E+09,9E+09,9E+09,9E+09,9E+09]];
	CONST robtarget Target_3310:=[[105.6,251.2,-49.1],[-0.00782265456170565,0.733639401003984,0.6574364462315,-0.171724647434841],[0,0,0,1],[9E+09,9E+09,9E+09,9E+09,9E+09,9E+09]];
	CONST robtarget Target_3320:=[[110.3,251,-50.3],[-0.00897562763950428,0.729208103588957,0.662348090658669,-0.17166824566439],[0,0,0,1],[9E+09,9E+09,9E+09,9E+09,9E+09,9E+09]];
	CONST robtarget Target_3330:=[[115,250.6,-51.6],[-0.0101362950557384,0.724712432235474,0.667264072240018,-0.171603624622428],[0,0,0,1],[9E+09,9E+09,9E+09,9E+09,9E+09,9E+09]];
	CONST robtarget Target_3340:=[[119.7,250.4,-52.8],[-0.0112925044941989,0.720199272482732,0.67213276921627,-0.171531419288889],[0,0,0,1],[9E+09,9E+09,9E+09,9E+09,9E+09,9E+09]];
	CONST robtarget Target_3350:=[[119.7,245.6,-51.8],[-0.0128588450933917,0.720115913737561,0.672557190492338,-0.170101576717661],[0,0,0,1],[9E+09,9E+09,9E+09,9E+09,9E+09,9E+09]];
	CONST robtarget Target_3360:=[[119.7,240.9,-50.8],[-0.0144181905769114,0.72005000024701,0.672956724338874,-0.168669381014636],[0,0,0,1],[9E+09,9E+09,9E+09,9E+09,9E+09,9E+09]];
	CONST robtarget Target_3370:=[[119.7,236.2,-49.8],[-0.015971633572572,0.719995604729686,0.673341915881814,-0.167218122246257],[0,0,0,1],[9E+09,9E+09,9E+09,9E+09,9E+09,9E+09]];
	CONST robtarget Target_3380:=[[119.7,231.5,-48.8],[-0.017522051639576,0.719944217002652,0.673713459494826,-0.1657814121254],[0,0,0,1],[9E+09,9E+09,9E+09,9E+09,9E+09,9E+09]];
	CONST robtarget Target_3390:=[[119.7,226.7,-47.9],[-0.0190720397614266,0.719887298952837,0.674080672462593,-0.164358696508904],[0,0,0,1],[9E+09,9E+09,9E+09,9E+09,9E+09,9E+09]];
	CONST robtarget Target_3400:=[[119.7,222,-47],[-0.0206141863419386,0.719849213890361,0.674425687869945,-0.162917636012926],[0,0,0,1],[9E+09,9E+09,9E+09,9E+09,9E+09,9E+09]];
	CONST robtarget Target_3410:=[[119.7,217.3,-46.1],[-0.0221522985735409,0.719817091465536,0.674758155864385,-0.161474646915544],[0,0,0,1],[9E+09,9E+09,9E+09,9E+09,9E+09,9E+09]];
	CONST robtarget Target_3420:=[[119.7,212.6,-45.2],[-0.0236886641589516,0.719786940489491,0.675078480097401,-0.160045784700893],[0,0,0,1],[9E+09,9E+09,9E+09,9E+09,9E+09,9E+09]];
	CONST robtarget Target_3430:=[[119.7,207.8,-44.3],[-0.025223237659445,0.719754635060129,0.675395034276378,-0.158614631312015],[0,0,0,1],[9E+09,9E+09,9E+09,9E+09,9E+09,9E+09]];
	CONST robtarget Target_3440:=[[119.7,203.1,-43.5],[-0.0267524651301361,0.719735227263147,0.675691775794042,-0.157181844912896],[0,0,0,1],[9E+09,9E+09,9E+09,9E+09,9E+09,9E+09]];
	CONST robtarget Target_3450:=[[119.7,198.4,-42.7],[-0.0282782545443338,0.719720645240234,0.675977312325804,-0.155747251518894],[0,0,0,1],[9E+09,9E+09,9E+09,9E+09,9E+09,9E+09]];
	CONST robtarget Target_3460:=[[119.7,193.7,-41.8],[-0.0298034665228329,0.719707226208557,0.676251912667609,-0.154326318364067],[0,0,0,1],[9E+09,9E+09,9E+09,9E+09,9E+09,9E+09]];
	CONST robtarget Target_3470:=[[119.7,189,-41.1],[-0.0313227011217989,0.719701525474739,0.676515916078243,-0.152888253036598],[0,0,0,1],[9E+09,9E+09,9E+09,9E+09,9E+09,9E+09]];
	CONST robtarget Target_3480:=[[119.7,184.2,-40.3],[-0.0328808379407684,0.719697403969569,0.676774392615492,-0.151429583357108],[0,0,0,1],[9E+09,9E+09,9E+09,9E+09,9E+09,9E+09]];
	CONST robtarget Target_3490:=[[119.7,179.5,-39.6],[-0.0343969212798386,0.719696439264827,0.677017651592734,-0.150003288456814],[0,0,0,1],[9E+09,9E+09,9E+09,9E+09,9E+09,9E+09]];
	CONST robtarget Target_3500:=[[119.7,174.8,-38.8],[-0.0359101121108122,0.719699125713495,0.677251057216981,-0.148575360655468],[0,0,0,1],[9E+09,9E+09,9E+09,9E+09,9E+09,9E+09]];
	CONST robtarget Target_3510:=[[119.7,170.1,-38.1],[-0.0374204463715451,0.719705234895391,0.677474850520684,-0.147145886689034],[0,0,0,1],[9E+09,9E+09,9E+09,9E+09,9E+09,9E+09]];
	CONST robtarget Target_3520:=[[119.7,165.3,-37.4],[-0.0389292896217268,0.719708346409807,0.677695848544467,-0.145714595642316],[0,0,0,1],[9E+09,9E+09,9E+09,9E+09,9E+09,9E+09]];
	CONST robtarget Target_3530:=[[119.7,160.6,-36.8],[-0.0404378111769494,0.719717853139121,0.677900787346707,-0.144296631335408],[0,0,0,1],[9E+09,9E+09,9E+09,9E+09,9E+09,9E+09]];
	CONST robtarget Target_3540:=[[119.7,155.9,-36.1],[-0.0419398630139701,0.719733141246756,0.678096934583651,-0.142862873377593],[0,0,0,1],[9E+09,9E+09,9E+09,9E+09,9E+09,9E+09]];
	CONST robtarget Target_3550:=[[119.7,151.2,-35.5],[-0.04344331380953,0.719748215733065,0.67828412552036,-0.141441965135516],[0,0,0,1],[9E+09,9E+09,9E+09,9E+09,9E+09,9E+09]];
	CONST robtarget Target_3560:=[[119.7,146.4,-34.9],[-0.044945509749326,0.719760119267005,0.678468776104705,-0.140019254808413],[0,0,0,1],[9E+09,9E+09,9E+09,9E+09,9E+09,9E+09]];
	CONST robtarget Target_3570:=[[119.7,141.7,-34.3],[-0.0464440772866591,0.719780190794116,0.678638852589163,-0.138595571292312],[0,0,0,1],[9E+09,9E+09,9E+09,9E+09,9E+09,9E+09]];
	CONST robtarget Target_3580:=[[119.7,137,-33.7],[-0.0479448372699026,0.719799803937581,0.67880042479814,-0.137184248820506],[0,0,0,1],[9E+09,9E+09,9E+09,9E+09,9E+09,9E+09]];
	CONST robtarget Target_3590:=[[119.7,132.3,-33.2],[-0.0494387596832467,0.71982411965525,0.678954212481979,-0.135757957985906],[0,0,0,1],[9E+09,9E+09,9E+09,9E+09,9E+09,9E+09]];
	CONST robtarget Target_3600:=[[119.7,127.5,-32.7],[-0.0509362308012004,0.719842507181339,0.6791053603599,-0.134343495477456],[0,0,0,1],[9E+09,9E+09,9E+09,9E+09,9E+09,9E+09]];
	CONST robtarget Target_3610:=[[119.7,122.8,-32.2],[-0.0524305493384612,0.7198680665055,0.679243054579513,-0.132928090060728],[0,0,0,1],[9E+09,9E+09,9E+09,9E+09,9E+09,9E+09]];
	CONST robtarget Target_3620:=[[119.7,118.1,-31.7],[-0.0539227905908445,0.719895285225862,0.679373134873898,-0.131511423747453],[0,0,0,1],[9E+09,9E+09,9E+09,9E+09,9E+09,9E+09]];
	CONST robtarget Target_3630:=[[119.7,113.4,-31.2],[-0.0554129551896327,0.719924020676598,0.679495748554978,-0.130093568425584],[0,0,0,1],[9E+09,9E+09,9E+09,9E+09,9E+09,9E+09]];
	CONST robtarget Target_3640:=[[119.7,108.6,-30.7],[-0.0569019629309244,0.719949270323902,0.679616191781681,-0.12867418794325],[0,0,0,1],[9E+09,9E+09,9E+09,9E+09,9E+09,9E+09]];
	CONST robtarget Target_3650:=[[119.7,103.9,-30.3],[-0.058387940861709,0.719980723710131,0.679724196561222,-0.127254164792231],[0,0,0,1],[9E+09,9E+09,9E+09,9E+09,9E+09,9E+09]];
	CONST robtarget Target_3660:=[[119.7,99.2,-29.9],[-0.0598776216216156,0.720011096866214,0.679824658385715,-0.125845638260513],[0,0,0,1],[9E+09,9E+09,9E+09,9E+09,9E+09,9E+09]];
	CONST robtarget Target_3670:=[[119.7,94.5,-29.5],[-0.0613655083938046,0.720042568279418,0.67991814027433,-0.124435914313536],[0,0,0,1],[9E+09,9E+09,9E+09,9E+09,9E+09,9E+09]];
	CONST robtarget Target_3680:=[[119.7,89.8,-29.1],[-0.0628515923557622,0.72007501831515,0.680004764514919,-0.123025060755081],[0,0,0,1],[9E+09,9E+09,9E+09,9E+09,9E+09,9E+09]];
	CONST robtarget Target_3690:=[[119.7,85,-28.8],[-0.064336655652234,0.720103899683729,0.680089342195864,-0.121612725614418],[0,0,0,1],[9E+09,9E+09,9E+09,9E+09,9E+09,9E+09]];
	CONST robtarget Target_3700:=[[119.7,80.3,-28.4],[-0.0658190780270005,0.720138044734531,0.680162517796056,-0.120199812308221],[0,0,0,1],[9E+09,9E+09,9E+09,9E+09,9E+09,9E+09]];
	CONST robtarget Target_3710:=[[119.7,75.6,-28.1],[-0.0672996627808184,0.720172832813,0.680229181677042,-0.118785969974019],[0,0,0,1],[9E+09,9E+09,9E+09,9E+09,9E+09,9E+09]];
	CONST robtarget Target_3720:=[[119.7,70.9,-27.8],[-0.0687850809253925,0.720206259937601,0.680288774358502,-0.117382874690421],[0,0,0,1],[9E+09,9E+09,9E+09,9E+09,9E+09,9E+09]];
	CONST robtarget Target_3730:=[[119.7,66.1,-27.6],[-0.0702696329912503,0.720236097011316,0.680346371155896,-0.1159782673443],[0,0,0,1],[9E+09,9E+09,9E+09,9E+09,9E+09,9E+09]];
	CONST robtarget Target_3740:=[[119.7,61.4,-27.3],[-0.0717448887914529,0.720272374985656,0.68039399227409,-0.114561738997581],[0,0,0,1],[9E+09,9E+09,9E+09,9E+09,9E+09,9E+09]];
	CONST robtarget Target_3750:=[[119.7,56.7,-27.1],[-0.0732253755943593,0.720307140577433,0.680434751151304,-0.113155720261464],[0,0,0,1],[9E+09,9E+09,9E+09,9E+09,9E+09,9E+09]];
	CONST robtarget Target_3760:=[[119.7,52,-26.8],[-0.0747115228913701,0.720340440006396,0.680468644477677,-0.111759843957285],[0,0,0,1],[9E+09,9E+09,9E+09,9E+09,9E+09,9E+09]];
	CONST robtarget Target_3770:=[[119.7,47.2,-26.6],[-0.0761895130311405,0.720371815338409,0.680501393526366,-0.110351525493748],[0,0,0,1],[9E+09,9E+09,9E+09,9E+09,9E+09,9E+09]];
	CONST robtarget Target_3780:=[[119.7,42.5,-26.5],[-0.0776727785581285,0.720405551888667,0.680523246637386,-0.108953618871318],[0,0,0,1],[9E+09,9E+09,9E+09,9E+09,9E+09,9E+09]];
	CONST robtarget Target_3790:=[[119.7,37.8,-26.3],[-0.0791469179971094,0.720440954411049,0.680540124134773,-0.107544111979611],[0,0,0,1],[9E+09,9E+09,9E+09,9E+09,9E+09,9E+09]];
	CONST robtarget Target_3800:=[[119.7,33.1,-26.2],[-0.0806272283124645,0.720474728202172,0.680550348761864,-0.106144424614581],[0,0,0,1],[9E+09,9E+09,9E+09,9E+09,9E+09,9E+09]];
	CONST robtarget Target_3810:=[[119.7,28.3,-26],[-0.0821066527591594,0.720504826362092,0.680558671847999,-0.104743433847213],[0,0,0,1],[9E+09,9E+09,9E+09,9E+09,9E+09,9E+09]];
	CONST robtarget Target_3820:=[[119.7,23.6,-25.9],[-0.083584041621182,0.720538427344595,0.680557491801351,-0.103342068196353],[0,0,0,1],[9E+09,9E+09,9E+09,9E+09,9E+09,9E+09]];
	CONST robtarget Target_3830:=[[119.7,18.9,-25.8],[-0.085059938553443,0.720571800799192,0.680550756587509,-0.101939955142535],[0,0,0,1],[9E+09,9E+09,9E+09,9E+09,9E+09,9E+09]];
	CONST robtarget Target_3840:=[[119.7,14.2,-25.8],[-0.0865428018846856,0.720603495890162,0.680537461381074,-0.100547047742977],[0,0,0,1],[9E+09,9E+09,9E+09,9E+09,9E+09,9E+09]];
	CONST robtarget Target_3850:=[[119.7,9.4,-25.7],[-0.0880162719808697,0.720632874639458,0.680523367054942,-0.0991430418519903],[0,0,0,1],[9E+09,9E+09,9E+09,9E+09,9E+09,9E+09]];
	CONST robtarget Target_3860:=[[119.7,4.7,-25.7],[-0.0894964456603955,0.720663942150709,0.680499152895289,-0.097748512043658],[0,0,0,1],[9E+09,9E+09,9E+09,9E+09,9E+09,9E+09]];
	CONST robtarget Target_3870:=[[124.4,0,-27],[-0.0913528683461587,0.718017695586607,0.683293600234328,-0.0959953027404928],[0,0,0,1],[9E+09,9E+09,9E+09,9E+09,9E+09,9E+09]];
	CONST robtarget Target_3880:=[[129.2,0,-28.2],[-0.0917373054742598,0.715270261770626,0.686169081147839,-0.0956279848560652],[0,0,0,1],[9E+09,9E+09,9E+09,9E+09,9E+09,9E+09]];
	CONST robtarget Target_3890:=[[133.9,0,-29.5],[-0.0921125499240875,0.712567117951155,0.688975803429609,-0.0952665883182135],[0,0,0,1],[9E+09,9E+09,9E+09,9E+09,9E+09,9E+09]];
	CONST robtarget Target_3900:=[[138.6,0,-30.8],[-0.0924865683539285,0.709851519696459,0.69177335542887,-0.0949035266859119],[0,0,0,1],[9E+09,9E+09,9E+09,9E+09,9E+09,9E+09]];
	CONST robtarget Target_3910:=[[143.3,0,-32.1],[-0.0928593068037467,0.707123828793847,0.694561333539825,-0.0945388483282778],[0,0,0,1],[9E+09,9E+09,9E+09,9E+09,9E+09,9E+09]];
	CONST robtarget Target_3920:=[[148,0,-33.4],[-0.0932307119159065,0.704384413548804,0.697339338662461,-0.0941726024858756],[0,0,0,1],[9E+09,9E+09,9E+09,9E+09,9E+09,9E+09]];
	CONST robtarget Target_3930:=[[152.7,0,-34.7],[-0.0936007309790527,0.701633648501588,0.700106976530759,-0.0938048392328268],[0,0,0,1],[9E+09,9E+09,9E+09,9E+09,9E+09,9E+09]];
	CONST robtarget Target_3940:=[[157.5,0,-36],[-0.0939771381189258,0.698813037467667,0.702922395405,-0.0934277379276937],[0,0,0,1],[9E+09,9E+09,9E+09,9E+09,9E+09,9E+09]];
	CONST robtarget Target_3950:=[[162.2,0,-37.2],[-0.094344197508849,0.69604049896328,0.705667895755247,-0.0930570636745044],[0,0,0,1],[9E+09,9E+09,9E+09,9E+09,9E+09,9E+09]];
	CONST robtarget Target_3960:=[[166.9,0,-38.5],[-0.0947097159521292,0.693257777098673,0.708401870260728,-0.0926850279580067],[0,0,0,1],[9E+09,9E+09,9E+09,9E+09,9E+09,9E+09]];
	CONST robtarget Target_3970:=[[171.6,0,-39.8],[-0.0950736437599509,0.690465268442623,0.711123947263166,-0.0923116837974231],[0,0,0,1],[9E+09,9E+09,9E+09,9E+09,9E+09,9E+09]];
	CONST robtarget Target_3980:=[[176.3,0,-41.1],[-0.0954359320949495,0.687663374245092,0.713833761472897,-0.0919370848378263],[0,0,0,1],[9E+09,9E+09,9E+09,9E+09,9E+09,9E+09]];
	CONST robtarget Target_3990:=[[181.1,0,-42.4],[-0.0958041866891989,0.684792599701108,0.716588201613234,-0.0915532769273203],[0,0,0,1],[9E+09,9E+09,9E+09,9E+09,9E+09,9E+09]];
	CONST robtarget Target_4000:=[[185.8,0,-43.7],[-0.0961630157502494,0.681972977364381,0.719272141432888,-0.0911763078059579],[0,0,0,1],[9E+09,9E+09,9E+09,9E+09,9E+09,9E+09]];
	CONST robtarget Target_4010:=[[190.5,0,-44.9],[-0.0965200633315447,0.679145206814953,0.721942756288174,-0.0907982493101276],[0,0,0,1],[9E+09,9E+09,9E+09,9E+09,9E+09,9E+09]];
	CONST robtarget Target_4020:=[[195.2,0,-46.2],[-0.0968752843818149,0.676309704729923,0.724599709208343,-0.0904191571474318],[0,0,0,1],[9E+09,9E+09,9E+09,9E+09,9E+09,9E+09]];
	CONST robtarget Target_4030:=[[199.9,0,-47.5],[-0.0972286348740366,0.673466890754551,0.727242670883721,-0.0900390874223009],[0,0,0,1],[9E+09,9E+09,9E+09,9E+09,9E+09,9E+09]];
	CONST robtarget Target_4040:=[[204.6,0,-48.8],[-0.0975800718352638,0.670617187149586,0.729871319888833,-0.0896580965888427],[0,0,0,1],[9E+09,9E+09,9E+09,9E+09,9E+09,9E+09]];
	CONST robtarget Target_4050:=[[209.3,0,-50.1],[-0.0979295533748152,0.667761018436432,0.732485342893241,-0.0892762414034031],[0,0,0,1],[9E+09,9E+09,9E+09,9E+09,9E+09,9E+09]];
	CONST robtarget Target_4060:=[[214.1,4.7,-51.4],[-0.0969419126319893,0.664341826293298,0.735585037755558,-0.0903706569783089],[0,0,0,1],[9E+09,9E+09,9E+09,9E+09,9E+09,9E+09]];
	CONST robtarget Target_4070:=[[214.1,9.4,-51.4],[-0.0956352507820257,0.663843336202951,0.73602677354098,-0.0918178218955898],[0,0,0,1],[9E+09,9E+09,9E+09,9E+09,9E+09,9E+09]];
	CONST robtarget Target_4080:=[[214.1,14.1,-51.4],[-0.0943048826559268,0.663330579630775,0.736472643001956,-0.093312257199492],[0,0,0,1],[9E+09,9E+09,9E+09,9E+09,9E+09,9E+09]];
	CONST robtarget Target_4090:=[[214.1,18.8,-51.5],[-0.0929667151175744,0.662811152057207,0.736920607127253,-0.0947976021851103],[0,0,0,1],[9E+09,9E+09,9E+09,9E+09,9E+09,9E+09]];
	CONST robtarget Target_4100:=[[214.1,23.5,-51.6],[-0.0916392101554855,0.662282314080756,0.737368414746666,-0.0962923286243821],[0,0,0,1],[9E+09,9E+09,9E+09,9E+09,9E+09,9E+09]];
	CONST robtarget Target_4110:=[[214.1,28.2,-51.7],[-0.0903476248802413,0.66175076707453,0.737813216726165,-0.0977490980979308],[0,0,0,1],[9E+09,9E+09,9E+09,9E+09,9E+09,9E+09]];
	CONST robtarget Target_4120:=[[214.1,32.9,-51.8],[-0.0890232355278324,0.661205404795119,0.738263427899601,-0.0992440790768353],[0,0,0,1],[9E+09,9E+09,9E+09,9E+09,9E+09,9E+09]];
	CONST robtarget Target_4130:=[[214.1,37.6,-52],[-0.0877005611737851,0.660651556753741,0.73871493975808,-0.10073911805688],[0,0,0,1],[9E+09,9E+09,9E+09,9E+09,9E+09,9E+09]];
	CONST robtarget Target_4140:=[[214.1,42.3,-52.1],[-0.0864225230900232,0.660093279955253,0.739162979927188,-0.102206156203186],[0,0,0,1],[9E+09,9E+09,9E+09,9E+09,9E+09,9E+09]];
	CONST robtarget Target_4150:=[[214.1,47,-52.3],[-0.0851034431169612,0.659522090614642,0.739617502834651,-0.103701328157192],[0,0,0,1],[9E+09,9E+09,9E+09,9E+09,9E+09,9E+09]];
	CONST robtarget Target_4160:=[[214.1,51.7,-52.5],[-0.0837945760408972,0.658940359613963,0.740072696951967,-0.105206818810331],[0,0,0,1],[9E+09,9E+09,9E+09,9E+09,9E+09,9E+09]];
	CONST robtarget Target_4170:=[[214.1,56.4,-52.8],[-0.0825219107000369,0.658355458149378,0.740526028980437,-0.10667438953096],[0,0,0,1],[9E+09,9E+09,9E+09,9E+09,9E+09,9E+09]];
	CONST robtarget Target_4180:=[[214.1,61.1,-53],[-0.0812168877925794,0.657755387238009,0.74098496061655,-0.108180200761296],[0,0,0,1],[9E+09,9E+09,9E+09,9E+09,9E+09,9E+09]];
	CONST robtarget Target_4190:=[[214.1,65.8,-53.3],[-0.0799139638073097,0.657145878750976,0.741445892179642,-0.10968610394734],[0,0,0,1],[9E+09,9E+09,9E+09,9E+09,9E+09,9E+09]];
	CONST robtarget Target_4200:=[[214.1,70.5,-53.5],[-0.0786209131429899,0.656524923359305,0.741908117772246,-0.111203065642386],[0,0,0,1],[9E+09,9E+09,9E+09,9E+09,9E+09,9E+09]];
	CONST robtarget Target_4210:=[[214.1,75.2,-53.8],[-0.0773566576912869,0.655902245050804,0.742370135670044,-0.112671088187645],[0,0,0,1],[9E+09,9E+09,9E+09,9E+09,9E+09,9E+09]];
